(* CODESYS project Lib.library
   Author: Sha
   Placeholder: Lib
   Title: Lib
   Version: 0.1.2
   DefaultNamespace: Lib
   Company: Terza-automation

Project tree, tasks and I/O mapping:
  libraries: CmpBitmapPool, * (System); Tc2_ModbusRTU, * (Beckhoff Automation GmbH); Tc2_Standard, * (Beckhoff Automation GmbH); Tc2_System, * (Beckhoff Automation GmbH); Tc2_Utilities, * (Beckhoff Automation GmbH); Tc3_Module, * (Beckhoff Automation GmbH)
  DUTs/
    data type Beckhoff_AI
    data type ModbusUnion
    data type RealWordUnion
    data type RTU_EM
    data type RTU_STS
    data type RTU_THT
  GVLs/
    global variables GVL
    global variables GVL_DataHalls
    global variables GVL_Electrical
    global variables GVL_EM
    global variables GVL_HW
    global variables GVL_PCS
    global variables GVL_SCS
    global variables GVL_STS
    global variables GVL_THT
  POUs/
    function block AccumDDHHMM [LD]
    function block AccumTimes [LD]
    function AI_OOR [ST]
    function block CAC_Analog [ST]
    function block CAC_Average [ST]
    function block CAC_Mirror [ST]
    function block FB_AI_Scaling [ST]
    function block FB_AO_Scaling [ST]
    program MAIN [ST]
    function block ModbusRTU_EM_Bell [ST]
    function block ModbusRTU_EM_Integra [ST]
    function block ModbusRTU_STS [ST]
    function block ModbusRTU_THT [ST]
    function block OneATS [ST]
    function block OneCRAH [ST]
    function block OneDI [ST]
    function block OneEnergyMeter [ST]
    function block OneFire_Suppr [ST]
    function block OneGen [ST]
    function block OneGLP [ST]
    function block OneIDF [ST]
    function block OneIsolator_Latch [LD]
    function block OnePDU [ST]
    function block OnePumpFF_Latch [LD]
    function block OneSpeed_Override [LD]
    function block OneSTS [ST]
    function block OneSTS_RTU [ST]
    function block OneSWBL [ST]
    function block OneTie_BRK [ST]
    function block OneUPS [ST]
    function block OneVSD_Latch [LD]
    function ReadModbusBool [ST]
    function ReadModbusReal [ST]
    function ReadModusTime [ST]
    function block WriteModbusBool [ST]
    function block WriteModbusReal [ST]
    function block WriteModbusWord [ST]
  Version/
    global variables Global_Version
  VISUs/
    visualisation AminCRAH
    text list CRAH_Isolator_Status
    text list CRAH_Status
    visualisation Dialog_CRAH
    visualisation Dialog_DP_Field
    visualisation Dialog_EnergyMeter
    visualisation Dialog_PDU
    visualisation Dialog_THT_Field
    text list Energy_Meters_Status
    text list Equipment_Status
    text list GLP_Available
    text list GLP_Status
    text list Leak_Detection_Fault
    visualisation Obj_Alarm_Equipment
    visualisation Obj_DP_Field
    visualisation Obj_Energy_Meter
    visualisation Obj_GLP_Avail
    visualisation Obj_GLP_Status
    visualisation Obj_Healthy_Failed_Field
    visualisation Obj_Leak_Detection
    visualisation Obj_PDU_Breaker
    visualisation Obj_PDU_Surge
    visualisation Obj_Terminal
    visualisation Obj_THT_Field
    text list PDU_Breaker_Status
    text list PDU_Surge_Status
  text list GlobalTextList
*)

// DUTs/Beckhoff_AI
TYPE Beckhoff_AI :
STRUCT
	rawValue   : WORD;
	OutOfRange : BOOL;
	Offline    : BOOL;
	Value      : REAL;

END_STRUCT
END_TYPE

// DUTs/ModbusUnion
TYPE ModbusUnion :
UNION
	realValue : REAL;
	longValue : DWORD;
	wordValue : ARRAY[1..2] OF WORD;
	timeValue : TIME;
END_UNION
END_TYPE

// DUTs/RealWordUnion
TYPE RealWordUnion :
UNION
	RealValue: REAL;
	UDINTValue: UDINT;
	WordArray: ARRAY[1..2] OF WORD;
END_UNION
END_TYPE

// DUTs/RTU_EM
TYPE RTU_EM :
STRUCT
	Status: WORD;
	Operating_Hrs: REAL;
	Energy: REAL;
	Volume: REAL;
	Supply_Temp: REAL;
	Return_Temp: REAL;
	Temp_Diff: REAL;
	CommsError: BOOL;
	CommsErrorCode: INT;	
END_STRUCT
END_TYPE

// DUTs/RTU_STS
TYPE RTU_STS :
STRUCT
	CommsError : BOOL;
	CommsErrorCode : INT;

	PRI_VA : REAL;
	PRI_VB : REAL;
	PRI_VC : REAL;
	OTP_VA : REAL;
	OTP_VB : REAL;
	OTP_VC : REAL;
	AMPSA : REAL;
	AMPSB : REAL;
	AMPSC : REAL;
	FREQ : REAL;
	SEC_VA : REAL;
	SEC_VB : REAL;
	SEC_VC : REAL;
	OTP_LOAD_A : REAL;
	OTP_LOAD_B : REAL;
	OTP_LOAD_C : REAL;
	COM_ALM : BOOL;
	OTP_KW_A : REAL;
	OTP_KW_B : REAL;
	OTP_KW_C : REAL;
	OTP_KVA_A : REAL;
	OTP_KVA_B : REAL;
	OTP_KVA_C : REAL;
	PF_A : REAL;
	PF_B : REAL;
	PF_C : REAL;

	OTP_BKR_OPN : BOOL;
	L1_INP_BKR_OPN : BOOL;
	L2_INP_BKR_OPN : BOOL;
	L1_BYP_BKR_TRP : BOOL;
	L2_BYP_BKR_TRP : BOOL;
	OTP_BKR_TRP : BOOL;
	L1_INP_BKR_TRP : BOOL;
	L2_INP_BKR_TRP : BOOL;
	FANS_FAIL : BOOL;
	
END_STRUCT
END_TYPE

// DUTs/RTU_THT
TYPE RTU_THT :
STRUCT
	Temp: REAL;
	RH: REAL;
	Temp_OOR : BOOL;
	RH_OOR : BOOL;
	CommsError : BOOL;
	CommsErrorCode : INT;	
END_STRUCT
END_TYPE

// GVLs/GVL
{attribute 'qualified_only'}
VAR_GLOBAL
	mb_Input_Coils    	:	ARRAY [0..511] OF BOOL;
	mb_Output_Coils 	:   ARRAY [0..511] OF BOOL;
 	mb_Input_Registers 	:   ARRAY [0..511] OF WORD;
 	mb_Output_Registers :   ARRAY [0..255] OF WORD;
	
	nInputCoilIndex: INT;
	nOutputCoilIndex: INT;
	nInputRegisterIndex: INT;
	nOutputRegisterIndex: INT;
END_VAR

// GVLs/GVL_DataHalls
{attribute 'qualified_only'}
VAR_GLOBAL CONSTANT
	StartInputCoilIndex_CRAH : INT := 0;			// uses 0-95
	StartInputCoilIndex_PDU : INT := 120;			// uses 120-295 
	StartInputCoilIndex_CAC : INT := 0;				// not used
	StartInputCoilIndex_IDF : INT := 310;           // uses 310-331
	StartInputCoilIndex_GLP : INT := 350;           // uses 350-361
	StartInputCoilIndex_ATS : INT := 370;           // uses 370-385
	StartInputCoilIndex_OtherDIs : INT := 400;		// uses 400-411
	StartInputCoilIndex_E_METER : INT := 420;		// uses 420-421
	StartInputCoilIndex_IO : INT := 430;			// uses 430-469
    StartInputCoilIndex_RTUStat : INT := 480;		// uses 480-495
	
	StartOutputCoilIndex_CRAH : INT := 0;			// uses 0-31
	StartOutputCoilIndex_PDU : INT := 0;			// not used
	StartOutputCoilIndex_CAC : INT := 80;			// uses 80-447
	StartOutputCoilIndex_OtherDIs : INT := 0;		// not used
	StartoutputCoilIndex_E_METER : INT := 0;		// not used
	StartoutputCoilIndex_IO : INT := 0;				// not used
	StartoutputCoilIndex_IDF : INT := 0;	        // not used
	StartoutputCoilIndex_GLP : INT := 0;	        // not used
	StartoutputCoilIndex_ATS : INT := 60;	        // uses 60-65
	StartOutputCoilIndex_RTUStat : INT := 0;	    // not used
	
	StartInputRegisterIndex_CRAH: INT := 0;			// uses 0-127
	StartInputRegisterIndex_PDU: INT := 0;			// not used
	StartInputRegisterIndex_CAC: INT := 0;			// not used
	StartInputRegisterIndex_OtherDIs : INT := 0;	// not used
	StartInputRegisterIndex_E_METER : INT := 128;	// uses 128-154
    StartInputRegisterIndex_IO : INT := 0;			// not used
	StartInputRegisterIndex_IDF : INT := 0;			// not used
	StartInputRegisterIndex_GLP : INT := 0;			// not used
	StartInputRegisterIndex_ATS : INT := 0;			// not used
	StartInputRegisterIndex_RTUStat : INT := 161;	// uses 161-176 
		
	StartOutputRegisterIndex_CRAH: INT := 0;		// not used
	StartOutputRegisterIndex_PDU: INT := 0;			// not used
	StartOutputRegisterIndex_CAC: INT := 0;			// uses 0-143
	StartOutputRegisterIndex_OtherDIs : INT := 0;	// not used
	StartoutputRegisterIndex_E_METER : INT := 0;	// not used
	StartoutputRegisterIndex_IO : INT := 0;			// not used
	StartoutputRegisterIndex_IDF : INT := 0;		// not used
	StartoutputRegisterIndex_GLP : INT := 0;		// not used
	StartoutputRegisterIndex_ATS : INT := 0;		// not used
	StartOutputRegisterIndex_RTUStat : INT := 0;	// not used
	


END_VAR

// GVLs/GVL_Electrical
{attribute 'qualified_only'}
VAR_GLOBAL CONSTANT
	StartInputCoilIndex_CRAH : INT := 0;			     // uses 0-29
	StartInputCoilIndex_SWBL : INT := 30;			     // uses 30-122 (third & fourth switchboards and STS overlap, but no system has these)
	StartInputCoilIndex_CAC : INT := 0;				     // not used
	StartInputCoilIndex_STS : INT := 98;			     // uses 98-225 no panel has STS and either GLP or ATS
	StartInputCoilIndex_GLP : INT := 210;          		 // uses 210-221
	StartInputCoilIndex_ATS : INT := 222;                // uses 222-244 no panel has ATS and GEN
	StartInputCoilIndex_GEN : INT := 238;			     // uses 238-247
	StartInputCoilIndex_UPS : INT := 248;			     // uses 248-262
	StartInputCoilIndex_TX : INT := 263;			     // uses 263-270
	StartInputCoilIndex_Fire_Suppr : INT := 273;		 // uses 273-296
	StartInputCoilIndex_OtherDIs : INT := 297;		     // uses 297-330
	StartInputCoilIndex_STSRTU : INT := 331;		     // uses 331-407
 	StartInputCoilIndex_IO : INT := 408;				 // uses 408-430
 	StartInputCoilIndex_RTUStat : INT := 431;		 	 // uses 431-440
	StartInputCoilIndex_Tie_BRK : INT := 450;            // uses 450-465
	StartInputCoilIndex_EMG_LIT : INT := 471;			 // uses 471-488
   
	StartOutputCoilIndex_CRAH : INT := 0;			     // uses 0-11
	StartOutputCoilIndex_SWBL : INT := 0;			     // not used
	StartOutputCoilIndex_CAC : INT := 23;			     // uses 23-52
	StartOutputCoilIndex_OtherDIs : INT := 0;		     // not used 
	StartOutputCoilIndex_GEN : INT := 0;	             // not used
	StartOutputCoilIndex_UPS : INT := 0;	             // not used
	StartOutputCoilIndex_TX : INT := 0;				     // not used
	StartOutputCoilIndex_Fire_Suppr : INT := 0;	         // not used
	StartOutputCoilIndex_ATS : INT := 20;	             // uses 20-22
	StartOutputCoilIndex_GLP : INT := 0;	      		 // not used
	StartOutputCoilIndex_Tie_BRK : INT := 0;	         // not used
	StartOutputCoilIndex_STS : INT := 12;	             // uses 12-19
	StartOutputCoilIndex_STSRTU : INT := 0;	             // not used
 	StartOutputCoilIndex_IO : INT := 0;				 	 // not used
 	StartOutputCoilIndex_RTUStat : INT := 0;			 // not used
	StartOutputCoilIndex_EMG_LIT : INT := 0;	         // not used 
	
	StartInputRegisterIndex_CRAH: INT := 0;			     // uses 0-46
	StartInputRegisterIndex_SWBL: INT := 0;			     // not used
	StartInputRegisterIndex_CAC: INT := 0;			     // not used
	StartInputRegisterIndex_OtherDIs : INT := 0;	     // not used
	StartInputRegisterIndex_GEN : INT := 0;			     // not used
	StartInputRegisterIndex_UPS : INT := 0;			     // not used
    StartInputRegisterIndex_TX : INT := 0;			     // not used
	StartInputRegisterIndex_Fire_Suppr : INT := 0;	     // not used
	StartInputRegisterIndex_ATS : INT := 0;			     // not used
	StartInputRegisterIndex_GLP : INT := 0;	    		 // not used
	StartInputRegisterIndex_Tie_BRK : INT := 0;	         // not used
	StartInputRegisterIndex_STS : INT := 0;			     // not used
	StartInputRegisterIndex_STSRTU : INT := 61;			 // uses 61-460
 	StartInputRegisterIndex_IO : INT := 0;				 // not used
 	StartInputRegisterIndex_RTUStat : INT := 47;		 // uses 47-56
	StartInputRegisterIndex_EMG_LIT : INT := 0;			 // not used
		
	StartOutputRegisterIndex_CRAH: INT := 0;		     // not used
	StartOutputRegisterIndex_SWBL: INT := 0;		     // not used
	StartOutputRegisterIndex_CAC: INT := 0;			     // uses 0-10
	StartOutputRegisterIndex_OtherDIs : INT := 0;	     // not used
	StartOutputRegisterIndex_GEN : INT := 0;			 // not used
	StartOutputRegisterIndex_UPS : INT := 0;			 // not used
	StartOutputRegisterIndex_TX : INT := 0;			     // not used
	StartOutputRegisterIndex_Fire_Suppr : INT := 0;	     // not used
	StartOutputRegisterIndex_ATS : INT := 0;		     // not used
	StartOutputRegisterIndex_GLP : INT := 0;			 // not used
	StartOutputRegisterIndex_Tie_BRK : INT := 0;		 // not used
	StartOutputRegisterIndex_STS : INT := 0;			 // not used
	StartOutputRegisterIndex_STSRTU : INT := 0;			 // not used
 	StartOutputRegisterIndex_IO : INT := 0;				 // not used
 	StartOutputRegisterIndex_RTUStat : INT := 0;		 // not used
	StartOutputRegisterIndex_EMG_LIT : INT := 0;	     // not used
	
END_VAR

// GVLs/GVL_EM
{attribute 'qualified_only'}
VAR_GLOBAL
	EM: ARRAY[1..5] OF RTU_EM;
END_VAR

// GVLs/GVL_HW
{attribute 'qualified_only'}
VAR_GLOBAL
	//Date and Time
    fbGetLocalSystemTime: FB_LocalSystemTime;
	sSystemDateTime : STRING;
	sSystemTime : STRING;
	sSystemDate : STRING;	

	// Coupler state - a UINT that should be 8 if its healthy
	CouplerStatus AT %I* : UINT;
	Term02Status AT %I* : WORD;
	Term03Status AT %I* : WORD;
	Term04Status AT %I* : WORD;
	Term05Status AT %I* : WORD;
	Term06Status AT %I* : WORD;
	Term07Status AT %I* : WORD;
	Term08Status AT %I* : WORD;
	Term09Status AT %I* : WORD;
	Term10Status AT %I* : WORD;
	Term11Status AT %I* : WORD;
	Term12Status AT %I* : WORD;
	Term13Status AT %I* : WORD;
	Term14Status AT %I* : WORD;
	Term15Status AT %I* : WORD;
	Term16Status AT %I* : WORD;
	Term17Status AT %I* : WORD;
	Term18Status AT %I* : WORD;
	Term19Status AT %I* : WORD;
	Term20Status AT %I* : WORD;
	Term21Status AT %I* : WORD;
	Term22Status AT %I* : WORD;
	Term23Status AT %I* : WORD;
	Term24Status AT %I* : WORD;
	Term25Status AT %I* : WORD;
	Term26Status AT %I* : WORD;
	Term27Status AT %I* : WORD;
	Term28Status AT %I* : WORD;
	Term29Status AT %I* : WORD;
	Term30Status AT %I* : WORD;
	Term31Status AT %I* : WORD;
	Term32Status AT %I* : WORD;
	Term33Status AT %I* : WORD;
	Term34Status AT %I* : WORD;
	Term35Status AT %I* : WORD;
	Term36Status AT %I* : WORD;
    Term37Status AT %I* : WORD;
    Term38Status AT %I* : WORD;
    Term39Status AT %I* : WORD;
    Term40Status AT %I* : WORD;
	
	// I/O module status
	CouplerOffline : BOOL;
	Term02Offline : BOOL;
	Term03Offline : BOOL;
	Term04Offline : BOOL;
	Term05Offline : BOOL;
	Term06Offline : BOOL;
	Term07Offline : BOOL;
	Term08Offline : BOOL;
	Term09Offline : BOOL;
	Term10Offline : BOOL;
	Term11Offline : BOOL;
	Term12Offline : BOOL;
	Term13Offline : BOOL;
	Term14Offline : BOOL;
	Term15Offline : BOOL;
	Term16Offline : BOOL;
	Term17Offline : BOOL;
	Term18Offline : BOOL;
	Term19Offline : BOOL;
	Term20Offline : BOOL;
	Term21Offline : BOOL;
	Term22Offline : BOOL;
	Term23Offline : BOOL;
	Term24Offline : BOOL;
	Term25Offline : BOOL;
	Term26Offline : BOOL;
	Term27Offline : BOOL;
	Term28Offline : BOOL;
	Term29Offline : BOOL;
	Term30Offline : BOOL;
	Term31Offline : BOOL;
	Term32Offline : BOOL;
	Term33Offline : BOOL;
	Term34Offline : BOOL;
	Term35Offline : BOOL;
	Term36Offline : BOOL;
	Term37Offline : BOOL;
	Term38Offline : BOOL;
	Term39Offline : BOOL;
	Term40Offline : BOOL;
END_VAR

// GVLs/GVL_PCS
{attribute 'qualified_only'}
VAR_GLOBAL
	StartInputCoilIndex_DI: 			INT:=0;		// hardwired DI state sent to OA	
	StartInputCoilIndex_DO: 			INT:=40;	// hardwired DO state sent to OA
	StartInputCoilIndex_TerminalStatus: INT:=50;	// module state sent to OA
	StartInputCoilIndex_AI: 			INT:=100;	// AI OutOfRange status sent to OA
	StartInputCoilIndex_Control:		INT:=200;	// boolean values for control sent by OA
	
	StartOutputCoilIndex_DO: 			INT:=0;		// OA demand for state of digital outputs
	StartOutputCoilIndex_Control:		INT:=200;	// boolean values for control sent to OA
	
	StartInputRegisterIndex_AI: 		INT:=0;		// hardwired AI states sent to OA (each sent as real, using two registers)
    StartInputRegisterIndex_AO:	        INT:=50;	// hardwired AI states sent to OA (each sent as real, using two registers)
	StartInputRegisterIndex_Control:	INT:=200;	// integer and real values for control sent by OA

	StartOutputRegisterIndex_AO: 		INT:=0;		// OA demand for states of analog outputs
	StartOutputRegisterIndex_Control:	INT:=200;	// integer and real values for control sent to OA
END_VAR

// GVLs/GVL_SCS
{attribute 'qualified_only'}
VAR_GLOBAL
	
	StartInputCoilIndex_DI: 			INT:=0;		// hardwired DI state sent to OA	
	StartInputCoilIndex_DO: 			INT:=40;	// hardwired DO state sent to OA
	StartInputCoilIndex_TerminalStatus: INT:=50;	// module state sent to OA
	StartInputCoilIndex_AI: 			INT:=100;	// AI OutOfRange status sent to OA
	StartInputCoilIndex_RTUStat:		INT:=150;	// RTU comms status 
	StartInputCoilIndex_Control:		INT:=200;	// boolean values for control sent by OA
	StartInputCoilIndex_E_Meter:		INT:=250;	// Energy meter comms status
	
	StartOutputCoilIndex_DO: 			INT:=0;		// OA demand for state of digital outputs
	StartOutputCoilIndex_RTUStat:		INT:= 0;	// not used
	StartOutputCoilIndex_Control:		INT:=200;	// boolean values for control sent to OA
	StartOutputCoilIndex_E_Meter:		INT:= 0;	// not used
	
	StartInputRegisterIndex_AI: 		INT:=0;		// hardwired AI states sent to OA (each sent as real, using two registers)
    StartInputRegisterIndex_AO:	        INT:=50;	// hardwired AI states sent to OA (each sent as real, using two registers)
	StartInputRegisterIndex_RTUStat:	INT:=150;	// RTU comms error codes 
	StartInputRegisterIndex_Control:	INT:=200;	// integer and real values for control sent by OA
	StartInputRegisterIndex_E_Meter:	INT:=250;	// Energy meter data 

	StartOutputRegisterIndex_AO: 		INT:=0;		// OA demand for states of analog outputs
	StartOutputRegisterIndex_RTUStat:	INT:= 0;	// not used
	StartOutputRegisterIndex_Control:	INT:=200;	// integer and real values for control sent to OA
	StartOutputRegisterIndex_E_Meter:	INT:= 0;	// not used

END_VAR

// GVLs/GVL_STS
{attribute 'qualified_only'}
VAR_GLOBAL
	STS : ARRAY [1..10] OF RTU_STS;
END_VAR

// GVLs/GVL_THT
{attribute 'qualified_only'}
VAR_GLOBAL
	THT : ARRAY [1..14] OF RTU_THT;
END_VAR

VAR_GLOBAL CONSTANT
	Temp_OOR_Min : REAL :=   0.0;
	Temp_OOR_Max : REAL :=  50.0;
	RH_OOR_Min   : REAL :=   0.0;
	RH_OOR_Max   : REAL := 100.0;
END_VAR

// Version/Global_Version
{attribute 'TcGenerated'}
{attribute 'no-analysis'}
{attribute 'linkalways'}
// This function has been automatically generated from the project information.
VAR_GLOBAL CONSTANT
	{attribute 'const_non_replaced'}
	stLibVersion_Lib : ST_LibVersion := (iMajor := 0, iMinor := 1, iBuild := 2, iRevision := 0, nFlags := 0, sVersion := '0.1.2');
END_VAR

// POUs/AccumDDHHMM
FUNCTION_BLOCK AccumDDHHMM
VAR_INPUT
	State: BOOL;
	Retentive: BOOL;
	Reset:BOOL;
END_VAR

VAR PERSISTENT
	Mins: WORD;
	Hrs:  WORD;
	Days: WORD;	
END_VAR
VAR
	DisplayTime: STRING;
	timer: TON;
	timerPT: TIME:= T#1M;
	StateToOff: F_TRIG;
END_VAR

VAR_TEMP
	displayTimeFormat: FB_FormatString;
END_VAR
VAR // added by the converter: edge detectors and wires of the graphical bodies
    _w1, _w2, _w3, _w4 : BOOL;
END_VAR

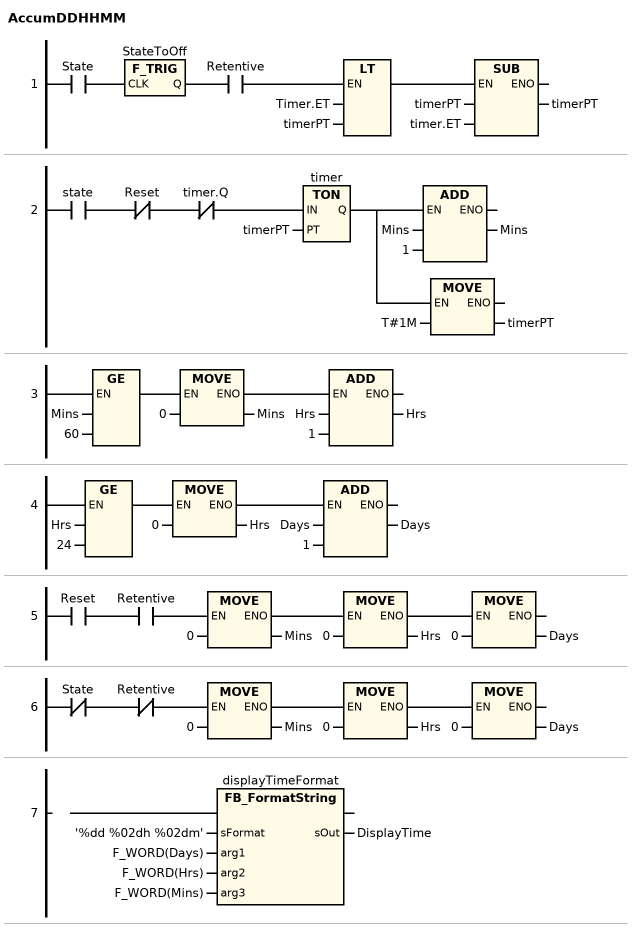
// NETWORK 1
StateToOff(CLK := State); // F_TRIG
IF StateToOff.Q AND Retentive AND Timer.ET < timerPT THEN timerPT := timerPT - timer.ET; END_IF

// NETWORK 2
timer(IN := state AND NOT Reset AND NOT timer.Q, PT := timerPT); // TON
IF timer.Q THEN Mins := Mins + 1; END_IF
IF timer.Q THEN timerPT := T#1M; END_IF

// NETWORK 3
_w1 := Mins >= 60;
IF _w1 THEN Mins := 0; END_IF
IF _w1 THEN Hrs := Hrs + 1; END_IF

// NETWORK 4
_w2 := Hrs >= 24;
IF _w2 THEN Hrs := 0; END_IF
IF _w2 THEN Days := Days + 1; END_IF

// NETWORK 5
_w3 := Reset AND Retentive;
IF _w3 THEN Mins := 0; END_IF
IF _w3 THEN Hrs := 0; END_IF
IF _w3 THEN Days := 0; END_IF

// NETWORK 6
_w4 := NOT State AND NOT Retentive;
IF _w4 THEN Mins := 0; END_IF
IF _w4 THEN Hrs := 0; END_IF
IF _w4 THEN Days := 0; END_IF

// NETWORK 7
displayTimeFormat(
    sFormat := '%dd %02dh %02dm',
    arg1 := F_WORD(Days),
    arg2 := F_WORD(Hrs),
    arg3 := F_WORD(Mins),
    sOut => DisplayTime); // FB_FormatString

END_FUNCTION_BLOCK

// POUs/AccumTimes
FUNCTION_BLOCK AccumTimes
VAR_INPUT
	State: BOOL;	
END_VAR

VAR PERSISTENT
	Num : WORD;
	ResetAccum: BOOL;

	cntOn: CTU;
	Accum: AccumDDHHMM;
	On: AccumDDHHMM;
	Off: AccumDDHHMM;
END_VAR

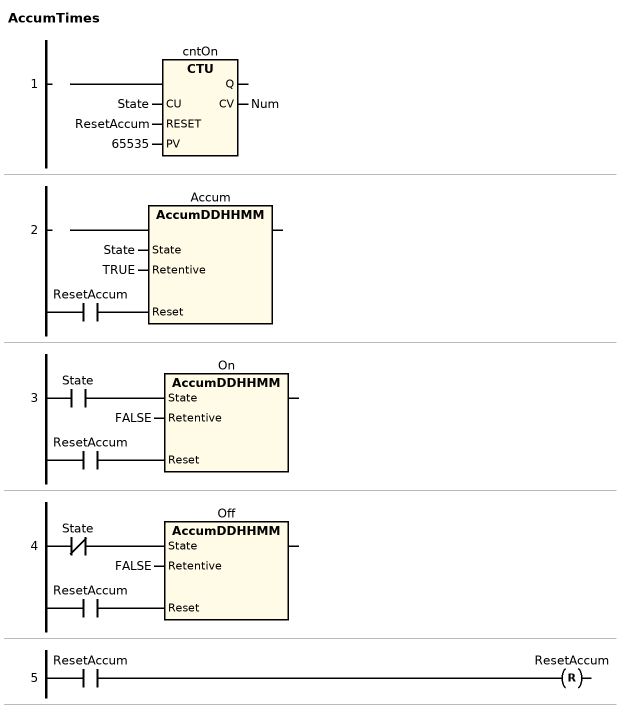
// NETWORK 1
cntOn(CU := State, RESET := ResetAccum, PV := 65535, CV => Num); // CTU

// NETWORK 2
Accum(State := State, Retentive := TRUE, Reset := ResetAccum); // AccumDDHHMM

// NETWORK 3
On(State := State, Retentive := FALSE, Reset := ResetAccum); // AccumDDHHMM

// NETWORK 4
Off(State := NOT State, Retentive := FALSE, Reset := ResetAccum); // AccumDDHHMM

// NETWORK 5
ResetAccum R= ResetAccum;

END_FUNCTION_BLOCK

// POUs/AI_OOR
FUNCTION AI_OOR : bool
VAR_INPUT
	Status: WORD;
END_VAR

// calculate whether the status for an analog input is indicating an error
// the error bit is the 7th bit of the status word
// access to bits is base 0, so the 7th bit is accessed with index 6

AI_OOR:= Status.6;

END_FUNCTION

// POUs/CAC_Analog
FUNCTION_BLOCK CAC_Analog
VAR_INPUT
	Value: REAL;
	OutOfRange : BOOL;
	Offline: BOOL;
END_VAR
VAR
	SetInclude: BOOL;
	SetExclude : BOOL;
	Excluded: BOOL;
	Alarm : BOOL;
	SetIncludeTrig: R_TRIG;
	SetExcludeTrig: R_TRIG;
END_VAR

VAR_TEMP
	i:INT;
	modbusReal: ModbusUnion;
END_VAR


i:= GVL.nOutputRegisterIndex;
modbusReal.realValue:= Value;
GVL.mb_Output_Registers[i+0]:= modbusReal.wordValue[1];
GVL.mb_Output_Registers[i+1]:= modbusReal.wordValue[2];
GVL.nOutputRegisterIndex:=i+2;

i:= GVL.nOutputCoilIndex;
GVL.mb_Output_Coils[i]:= OutOfRange;
GVL.mb_Output_Coils[i+1]:= Offline;

SetIncludeTrig(CLK:= SetInclude);
IF SetIncludeTrig.Q THEN 
	GVL.mb_Output_Coils[i+2]:= TRUE;
ELSIF SetInclude AND GVL.mb_Output_Coils[i+2] = FALSE THEN
 	SetInclude:=FALSE;
END_IF


SetExcludeTrig(CLK:=SetExclude);
IF SetExcludeTrig.Q THEN 
	GVL.mb_Output_Coils[i+3]:= TRUE;	
ELSIF SetExclude AND GVL.mb_Output_Coils[i+3]= FALSE THEN 
	SetExclude:=FALSE;
END_IF


Excluded:= GVL.mb_Output_Coils[i+4];
Alarm:= GVL.mb_Output_Coils[i+5];

GVL.nOutputCoilIndex:= i + 6;

END_FUNCTION_BLOCK

// POUs/CAC_Average
FUNCTION_BLOCK CAC_Average
VAR_INPUT
END_VAR
VAR_OUTPUT
END_VAR
VAR
	Value: REAL;
	Alarm: BOOL;
	OutOfRange: BOOL;
	Offline: BOOL;
END_VAR

VAR_TEMP
	i: INT;
	modbusReal: ModbusUnion;
END_VAR


i:= GVL.nOutputRegisterIndex;
modbusReal.wordValue[1]:= GVL.mb_Output_Registers[i+0];
modbusReal.wordValue[2]:= GVL.mb_Output_Registers[i+1];

Value:= modbusReal.realValue;
GVL.nOutputRegisterIndex:= i+2;


i:= GVL.nOutputCoilIndex;
OutOfRange:= FALSE;
Offline:= GVL.mb_Output_Coils[i+0];
Alarm:= GVL.mb_Output_Coils[i+1];
GVL.nOutputCoilIndex:= i+2;

END_FUNCTION_BLOCK

// POUs/CAC_Mirror
FUNCTION_BLOCK CAC_Mirror
VAR
	Value: REAL;
	OutOfRange: BOOL;
	Offline: BOOL;
	SetInclude: BOOL;
	SetExclude: BOOL;
	Excluded: BOOL;
	Alarm: BOOL;
	SetIncludeTrig: R_TRIG;
	SetExcludeTrig: R_TRIG;
END_VAR

VAR_TEMP
	i:INT;
	modbusReal: ModbusUnion;
END_VAR


i:= GVL.nOutputRegisterIndex;
modbusReal.wordValue[1]:= GVL.mb_Output_Registers[i+0];
modbusReal.wordValue[2]:= GVL.mb_Output_Registers[i+1];
Value:= modbusReal.realValue;
GVL.nOutputRegisterIndex:= i+2;

i:= GVL.nOutputCoilIndex;
OutOfRange:= GVL.mb_Output_Coils[i+0];
Offline:= GVL.mb_Output_Coils[i+1];

SetIncludeTrig(CLK:=SetInclude);

IF SetIncludeTrig.Q THEN 
	GVL.mb_Output_Coils[i+2] := TRUE;
ELSIF SetInclude AND GVL.mb_Output_Coils[i+2]= FALSE THEN 
	SetInclude:= FALSE;
END_IF

SetExcludeTrig(CLK:= SetExclude);
	
IF SetExcludeTrig.Q THEN 
	GVL.mb_Output_Coils[i+3] := TRUE;
ELSIF SetExclude AND GVL.mb_Output_Coils[i+3]= FALSE THEN 
	SetExclude:= FALSE;
END_IF


Excluded:= GVL.mb_Output_Coils[i+4];
Alarm:= GVL.mb_Output_Coils[i+5];
GVL.nOutputCoilIndex:= i+6;

END_FUNCTION_BLOCK

// POUs/FB_AI_Scaling
FUNCTION_BLOCK FB_AI_Scaling
VAR_INPUT
	I_Input: INT;
	I_Input_Min:  REAL :=0;
	I_Input_Max:  REAL :=100;
	I_Output_Min: REAL :=0;
	I_Output_Max: REAL :=3;
END_VAR
VAR_OUTPUT
	O_Output:REAL;
	O_Error:BOOL;	
END_VAR
VAR
	L_Input:INT;
END_VAR

VAR_TEMP
	i:INT;
	modbusReal: ModbusUnion;
END_VAR


IF I_Input_Max <> 0 AND I_Output_Max <> 0 THEN 
	IF I_Input_Min <= I_Input_Max THEN 
		L_Input:=I_Input;
		O_Output:= ((I_Output_Max - I_Output_Min) / (I_Input_Max - I_Input_Min) * (I_input - I_Input_Min) + I_Output_Min);
		O_Error:=FALSE;
	ELSE
		I_Input:= L_Input;	
	END_IF
ELSE
	O_Error:=TRUE;
END_IF


i:=GVL.nInputRegisterIndex;
modbusReal.realValue:= O_Output;
GVL.mb_Input_Registers[i+0]:= modbusReal.wordValue[1];
GVL.mb_Input_Registers[i+1]:= modbusReal.wordValue[2];
GVL.nInputRegisterIndex:=i+2;

END_FUNCTION_BLOCK

// POUs/FB_AO_Scaling
FUNCTION_BLOCK FB_AO_Scaling
VAR_INPUT
	I_Input:REAL;
	I_Input_Min:REAL:=0;
	I_Input_Max:REAL:=100;
	I_Output_Min:REAL :=0;
	I_Output_Max:REAL :=0;
END_VAR

VAR_OUTPUT
	O_Output: INT;
	O_Error: BOOL;
END_VAR

VAR
	L_Input:REAL;
END_VAR

VAR_TEMP
	i:INT;
	modbusReal: ModbusUnion;
END_VAR


IF I_Input_Max <> 0 AND I_Output_Max <> 0 THEN 
	IF I_Input <=I_Input_Max THEN 	
		L_Input:= I_Input;
		O_Output:= REAL_TO_INT((I_Output_Max - I_Output_Min) / (I_Input_Max - I_Input_Min) * (I_input - I_Input_Min) + I_Output_Min);
		O_Error:= FALSE;	
	ELSE
		I_Input:= L_Input;	
	END_IF
ELSE	
	O_Error:= TRUE;
END_IF

i:= GVL.nInputRegisterIndex;
modbusReal.realValue := L_Input;
GVL.mb_Input_Registers[i+0] := modbusReal.WordValue[1];
GVL.mb_Input_Registers[i+1] := modbusReal.WordValue[2];
GVL.nInputRegisterIndex := i+2;

END_FUNCTION_BLOCK

// POUs/MAIN
PROGRAM MAIN
VAR
END_VAR

END_PROGRAM

// POUs/ModbusRTU_EM_Bell
FUNCTION_BLOCK ModbusRTU_EM_Bell
VAR_INPUT
	MB_FirstUnitID: BYTE;
	MB_LastUnitID:  BYTE;
	EM_First: INT := 1;
END_VAR
VAR_OUTPUT
END_VAR
VAR
END_VAR

END_FUNCTION_BLOCK

// POUs/ModbusRTU_EM_Integra
FUNCTION_BLOCK ModbusRTU_EM_Integra
VAR_INPUT
	MB_FirstUnitID: BYTE;
	MB_LastUnitID: BYTE;
	EM_First: INT := 1;
END_VAR

VAR
	ModbusTerm: ModbusRtuMaster_KL6x22B;
	
	MB_UnitID : BYTE := 0;
	MB_Address : WORD := 0;
	MB_Quantity : WORD := 2;
	MB_ReadData : ModbusUnion;

	MB_TrigRead : BOOL := FALSE;
	MB_CommState: (TRIGGER, TRIGGERED, WAIT_RESPONSE, SETUP_NEXT_MESSAGE) := TRIGGER;
	tmrDelay: TON;
END_VAR


VAR CONSTANT
	MODBUS_DELAY : TIME := T#100MS;
END_VAR

VAR	
	EMNum: INT;
	MessageNum: INT;
END_VAR

IF (MB_UnitID < MB_FirstUnitID) THEN
	MB_UnitID := MB_FirstUnitID;
	EMNum := EM_First;
	MessageNum := 1;
	MB_Address := 0;
END_IF

IF (MB_UnitID > MB_LastUnitID) THEN
	MB_UnitID := MB_FirstUnitID;
	EMNum := EM_First;
	MessageNum := 1;
	MB_Address := 0;
END_IF

ModbusTerm.ReadRegs(
	UnitID:= MB_UnitID, 
	Quantity:= MB_Quantity, 
	MBAddr:= MB_Address, 
	cbLength:= SIZEOF(MB_ReadData), 
	pMemoryAddr:= ADR(MB_ReadData), 
	Execute:= MB_TrigRead, 
	Timeout:= T#1S, 
	BUSY=> , 
	Error=> , 
	ErrorID=> , 
	cbRead=> );
	
	
CASE MB_CommState OF
	TRIGGER:
		tmrDelay(IN:=TRUE, PT:=MODBUS_DELAY);
		IF tmrDelay.Q THEN
			MB_TrigRead := TRUE;
			MB_CommState := TRIGGERED;
		END_IF

	TRIGGERED:
		tmrDelay(IN:=FALSE, PT:=MODBUS_DELAY);
		MB_TrigRead := FALSE;
		MB_CommState := WAIT_RESPONSE;

	WAIT_RESPONSE:
		IF NOT ModbusTerm.BUSY THEN
			GVL_EM.EM[EMNum].CommsError     := ModbusTerm.Error;
			GVL_EM.EM[EMNum].CommsErrorCode := ModbusTerm.ErrorId;
			IF NOT ModbusTerm.Error THEN
				IF MessageNum = 1 THEN
					GVL_EM.EM[EMNum].Status := MB_ReadData.wordValue[2];
				ELSIF MessageNum = 2 THEN
					GVL_EM.EM[EMNum].Operating_Hrs := MB_ReadData.realValue;
				ELSIF MessageNum = 3 THEN
					GVL_EM.EM[EMNum].Energy := MB_ReadData.realValue;
				ELSIF MessageNum = 4 THEN
					GVL_EM.EM[EMNum].Volume := MB_ReadData.realValue;
				ELSIF MessageNum = 5 THEN
					GVL_EM.EM[EMNum].Supply_Temp := MB_ReadData.realValue;
				ELSIF MessageNum = 6 THEN
					GVL_EM.EM[EMNum].Return_Temp := MB_ReadData.realValue;
				ELSIF MessageNum = 7 THEN
					GVL_EM.EM[EMNum].Temp_Diff := MB_ReadData.realValue;
 				END_IF
 
			END_IF
			
			MB_CommState := SETUP_NEXT_MESSAGE;
		END_IF

	SETUP_NEXT_MESSAGE:
		MessageNum := MessageNum + 1;
		IF MessageNum > 7 THEN
			MessageNum := 1;
			MB_UnitID := MB_UnitID + 1;
			EMNum := EMNum + 1;
		END_IF

		IF MessageNum = 1 THEN
			MB_Address := 0;	// read status in word 2
		ELSIF MessageNum = 2 THEN
			MB_Address := 6;	// read operating hours
		ELSIF MessageNum = 3 THEN
			MB_Address := 100;	// read energy
		ELSIF MessageNum = 4 THEN
			MB_Address := 200;	// read volume
		ELSIF MessageNum = 5 THEN
			MB_Address := 800;	// read supply temperature
		ELSIF MessageNum = 6 THEN
			MB_Address := 810;	// read return temperature
		ELSIF MessageNum = 7 THEN
			MB_Address := 820;	// read temperature difference
		END_IF
	
		MB_CommState := TRIGGER;
END_CASE

END_FUNCTION_BLOCK

// POUs/ModbusRTU_STS
FUNCTION_BLOCK ModbusRTU_STS
VAR_INPUT
	MB_FirstUnitID: BYTE;
	MB_LastUnitID: BYTE;
END_VAR
VAR_OUTPUT
END_VAR
VAR
	ModbusTerm: ModbusRtuMaster_KL6x22B;
	
	MB_UnitID : BYTE := 0;
	MB_ReadData : ARRAY[1..71] OF WORD;

	MB_TrigRead : BOOL := FALSE;
	MB_CommState: (TRIGGER, TRIGGERED, WAIT_RESPONSE, SETUP_NEXT_MESSAGE) := TRIGGER;
	tmrDelay: TON;
END_VAR
	
VAR	
	STSNum: INT;
END_VAR


VAR CONSTANT
	MB_Address : WORD := 1;
	MB_Quantity : WORD := 71;

	MODBUS_DELAY : TIME := T#10MS;
END_VAR

IF (MB_UnitID < MB_FirstUnitID) THEN
	MB_UnitID := MB_FirstUnitID;
	STSNum := 1;
END_IF

IF (MB_UnitID > MB_LastUnitID) THEN
	MB_UnitID := MB_FirstUnitID;
	STSNum := 1;
END_IF

ModbusTerm.ReadRegs (
	UnitID:= MB_UnitID, 
	Quantity:= MB_Quantity, 
	MBAddr:= MB_Address - 1, 
	cbLength:= SIZEOF(MB_ReadData), 
	pMemoryAddr:= ADR(MB_ReadData), 
	Execute:= MB_TrigRead, 
	Timeout:= T#1S, 
	BUSY=> , 
	Error=> , 
	ErrorID=> , 
	cbRead=> );
	
CASE MB_CommState OF
	TRIGGER:
		tmrDelay(IN:=TRUE, PT:=MODBUS_DELAY);
		IF tmrDelay.Q THEN
			MB_TrigRead := TRUE;
			MB_CommState := TRIGGERED;
		END_IF

	TRIGGERED:
		tmrDelay(IN:=FALSE, PT:=MODBUS_DELAY);
		MB_TrigRead := FALSE;
		MB_CommState := WAIT_RESPONSE;

	WAIT_RESPONSE:
		IF NOT ModbusTerm.BUSY THEN
			GVL_STS.STS[STSNum].CommsError     := ModbusTerm.Error;
			GVL_STS.STS[STSNum].CommsErrorCode := ModbusTerm.ErrorId;
			IF NOT ModbusTerm.Error THEN
//				IF MessageNum = 1 THEN	// extracts the values in 13 registers #1-13
					GVL_STS.STS[STSNum].PRI_VA := WORD_TO_REAL(MB_ReadData[1]);
					GVL_STS.STS[STSNum].PRI_VB := WORD_TO_REAL(MB_ReadData[2]);
					GVL_STS.STS[STSNum].PRI_VC := WORD_TO_REAL(MB_ReadData[3]);
					GVL_STS.STS[STSNum].OTP_VA := WORD_TO_REAL(MB_ReadData[4]);
					GVL_STS.STS[STSNum].OTP_VB := WORD_TO_REAL(MB_ReadData[5]);
					GVL_STS.STS[STSNum].OTP_VC := WORD_TO_REAL(MB_ReadData[6]);
					GVL_STS.STS[STSNum].AMPSA  := WORD_TO_REAL(MB_ReadData[7]);
					GVL_STS.STS[STSNum].AMPSB  := WORD_TO_REAL(MB_ReadData[8]);
					GVL_STS.STS[STSNum].AMPSC  := WORD_TO_REAL(MB_ReadData[9]);
					GVL_STS.STS[STSNum].FREQ   := WORD_TO_REAL(MB_ReadData[10]);
					GVL_STS.STS[STSNum].SEC_VA := WORD_TO_REAL(MB_ReadData[11]);
					GVL_STS.STS[STSNum].SEC_VB := WORD_TO_REAL(MB_ReadData[12]);
					GVL_STS.STS[STSNum].SEC_VC := WORD_TO_REAL(MB_ReadData[13]);

//				ELSIF MessageNum = 2 THEN	// extracts the values in 3 registers #17-19
					GVL_STS.STS[STSNum].OTP_LOAD_A := WORD_TO_REAL(MB_ReadData[17]);
					GVL_STS.STS[STSNum].OTP_LOAD_B := WORD_TO_REAL(MB_ReadData[18]);
					GVL_STS.STS[STSNum].OTP_LOAD_C := WORD_TO_REAL(MB_ReadData[19]);

//				ELSIF MessageNum = 3 THEN	// extracts the alarms - 4 registers #41-44
					// common alarm is bit 15 of register 41
					GVL_STS.STS[STSNum].COM_ALM :=MB_ReadData[41].15;
					// other alarms of interest are in register 43 
					GVL_STS.STS[STSNum].OTP_BKR_OPN    := MB_ReadData[43].0;
					GVL_STS.STS[STSNum].L1_INP_BKR_OPN := MB_ReadData[43].1;
					GVL_STS.STS[STSNum].L2_INP_BKR_OPN := MB_ReadData[43].2;
					GVL_STS.STS[STSNum].L1_BYP_BKR_TRP := MB_ReadData[43].3;
					GVL_STS.STS[STSNum].L2_BYP_BKR_TRP := MB_ReadData[43].4;
					GVL_STS.STS[STSNum].OTP_BKR_TRP    := MB_ReadData[43].5;
					GVL_STS.STS[STSNum].L1_INP_BKR_TRP := MB_ReadData[43].6;
					GVL_STS.STS[STSNum].L2_INP_BKR_TRP := MB_ReadData[43].7;
					GVL_STS.STS[STSNum].FANS_FAIL      := MB_ReadData[43].8;

//				ELSIF MessageNum = 4 THEN	// extracts the values in 6 registers #56-61
					GVL_STS.STS[STSNum].OTP_KW_A  := WORD_TO_REAL(MB_ReadData[56]) / 10.0;
					GVL_STS.STS[STSNum].OTP_KW_B  := WORD_TO_REAL(MB_ReadData[57]) / 10.0;
					GVL_STS.STS[STSNum].OTP_KW_C  := WORD_TO_REAL(MB_ReadData[58]) / 10.0;
					GVL_STS.STS[STSNum].OTP_KVA_A := WORD_TO_REAL(MB_ReadData[59]) / 10.0;
					GVL_STS.STS[STSNum].OTP_KVA_B := WORD_TO_REAL(MB_ReadData[60]) / 10.0;
					GVL_STS.STS[STSNum].OTP_KVA_C := WORD_TO_REAL(MB_ReadData[61]) / 10.0;

//				ELSIF MessageNum = 5 THEN	// extracts the values in 3 registers #69-71
					GVL_STS.STS[STSNum].PF_A := WORD_TO_REAL(MB_ReadData[69]) / 100.0;
					GVL_STS.STS[STSNum].PF_B := WORD_TO_REAL(MB_ReadData[70]) / 100.0;
					GVL_STS.STS[STSNum].PF_C := WORD_TO_REAL(MB_ReadData[71]) / 100.0;
// 				END_IF
 			END_IF
			
			MB_CommState := SETUP_NEXT_MESSAGE;
		END_IF

	SETUP_NEXT_MESSAGE:
		MB_UnitID := MB_UnitID + 1;
		STSNum := STSNum + 1;
	
		MB_CommState := TRIGGER;
END_CASE

END_FUNCTION_BLOCK

// POUs/ModbusRTU_THT
FUNCTION_BLOCK ModbusRTU_THT
VAR_INPUT
	MB_FirstUnitID: BYTE;
	MB_LastUnitID: BYTE;
END_VAR
VAR_OUTPUT
END_VAR
VAR
	ModbusTerm: ModbusRtuMasterV2_KL6x22B;
	
	MB_UnitID:   BYTE := 0;
	MB_Address:  WORD := 25;
	MB_Quantity: WORD := 4;
	MB_ReadData: ARRAY[1..2] OF ModbusUnion;
	
	MB_TrigRead: BOOL :=FALSE;
	MB_CommState: (TRIGGER, TRIGGERED, WAIT_RESPONSE):=TRIGGER;
	tmrDelay: TON;
END_VAR

IF MB_UnitID < MB_FirstUnitID THEN 
	MB_UnitID:= MB_FirstUnitID;
END_IF

IF MB_UnitID > MB_LastUnitID THEN 
	MB_UnitID:= MB_FirstUnitID;
END_IF

ModbusTerm.ReadRegs(
	UnitID:= MB_UnitID, 
	Quantity:= MB_Quantity, 
	MBAddr:= MB_Address, 
	cbLength:= SIZEOF(MB_ReadData), 
	pMemoryAddr:= ADR(MB_ReadData),  
	Execute:= MB_TrigRead, 
	Timeout:= T#2S, 
	BUSY=> , 
	Error=> , 
	ErrorId=> , 
	cbRead=> );
	
CASE MB_CommState OF 
	TRIGGER:
		tmrDelay(in:=TRUE, PT:=T#1S);
		IF tmrDelay.Q THEN
			MB_TrigRead:=TRUE;
			MB_CommState:=TRIGGERED;
		END_IF
		
	TRIGGERED:
		tmrDelay(in:=FALSE, PT:=T#1S);
		MB_TrigRead:=FALSE;
		MB_CommState:=WAIT_RESPONSE;
		
	WAIT_RESPONSE:
		IF NOT ModbusTerm.BUSY THEN 
			GVL_THT.THT[MB_UnitID].CommsError:= ModbusTerm.Error;
			GVL_THT.THT[MB_UnitID].CommsErrorCode:= ModbusTerm.ErrorId;
			
			IF NOT ModbusTerm.Error THEN 
				GVL_THT.THT[MB_UnitID].Temp:= MB_ReadData[1].realValue;
				GVL_THT.THT[MB_UnitID].RH  := MB_ReadData[2].realValue;
				
				
				GVL_THT.THT[MB_UnitID].Temp_OOR:= (GVL_THT.THT[MB_UnitID].Temp < GVL_THT.Temp_OOR_Min) OR 
												  (GVL_THT.THT[MB_UnitID].Temp > GVL_THT.Temp_OOR_Max);
												  
				GVL_THT.THT[MB_UnitID].Rh_OOR:= (GVL_THT.THT[MB_UnitID].RH < GVL_THT.RH_OOR_Min) OR 
												(GVL_THT.THT[MB_UnitID].RH > GVL_THT.RH_OOR_Max);		   
				
			END_IF
		
			MB_UnitID := MB_UnitID + 1;
			MB_CommState := TRIGGER;
	
		END_IF
END_CASE

END_FUNCTION_BLOCK

// POUs/OneATS
FUNCTION_BLOCK OneATS
VAR_INPUT
	ATS_Avai: BOOL;
	ATS_Avai_Offline : BOOL;
	ATS_SP1 : BOOL;
	ATS_SP1_Offline : BOOL;
	ATS_SP2 : BOOL;
	ATS_SP2_Offline : BOOL;
	ATS_SP0 : BOOL;
	ATS_SP0_Offline : BOOL;
END_VAR
VAR_OUTPUT
	
	Net_Priority : BOOL;
	Source_Priority : BOOL;
	Inhibited: BOOL;
	
END_VAR

VAR_TEMP
	i: INT;
END_VAR

i := GVL.nInputCoilIndex;

GVL.mb_Input_Coils[i+0] := ATS_Avai;
GVL.mb_Input_Coils[i+1] := ATS_Avai_Offline;

GVL.mb_Input_Coils[i+2] := ATS_SP1;
GVL.mb_Input_Coils[i+3] := ATS_SP1_Offline;

GVL.mb_Input_Coils[i+4] := ATS_SP2;
GVL.mb_Input_Coils[i+5] := ATS_SP2_Offline;

GVL.mb_Input_Coils[i+6] := ATS_SP0;
GVL.mb_Input_Coils[i+7] := ATS_SP0_Offline;

GVL.nInputCoilIndex := i + 8;

i:= GVL.nOutputCoilIndex;

Net_Priority := GVL.mb_Output_Coils[i+0];
Source_Priority :=  GVL.mb_Output_Coils[i+1];
Inhibited := GVL.mb_Output_Coils[i+2];

GVL.nOutputCoilIndex := i +3;

END_FUNCTION_BLOCK

// POUs/OneCRAH
FUNCTION_BLOCK OneCRAH
VAR_INPUT
	Running: BOOL;
	Alarm: BOOL;
	Iso1_1_Sts: BOOL;
	Iso1_2_Sts: BOOL;
	Offline: BOOL;	
END_VAR

VAR_OUTPUT
	Enable: BOOL;	
END_VAR

VAR PERSISTENT
	Maintenance: BOOL;
	Inhibited: BOOL;
	HOA: WORD;
	Run: AccumTimes;
	Alm: AccumTimes;
	Ena: AccumTimes;
END_VAR

VAR_TEMP
	i: INT;
	modbusReal: ModbusUnion; 
END_VAR

Run(State:= Running);
Alm(State:= Alarm);
Ena(State:= Enable);

i:= GVL.nInputCoilIndex;

GVL.mb_Input_Coils[i+0] :=  Running;
GVL.mb_Input_Coils[i+1] :=  Alarm;
GVL.mb_Input_Coils[i+2] :=  Offline;
GVL.mb_Input_Coils[i+3] :=  Iso1_1_Sts;
GVL.mb_Input_Coils[i+4] :=  Iso1_2_Sts;

GVL.nInputCoilIndex := i + 5;


i:=GVL.nOutputCoilIndex;

Enable:= GVL.mb_Output_Coils[i+0];
Inhibited:= GVL.mb_Output_Coils[i+1];

GVL.nOutputCoilIndex:= i + 2;

i:= GVL.nInputRegisterIndex;
GVL.mb_Input_Registers[i+0]:= HOA;
GVL.mb_Input_Registers[i+1]:= Run.Num;


modbusReal.realValue:= WORD_TO_REAL(Run.Accum.Days) * 24.0 +
					   WORD_TO_REAL(Run.Accum.Hrs) * 1.0 + 
					   WORD_TO_REAL(Run.Accum.Mins) / 60.0;

GVL.mb_Input_Registers[i+2]:= modbusReal.wordValue[1];
GVL.mb_Input_Registers[i+3]:= modbusReal.wordValue[2];	

modbusReal.realValue:= WORD_TO_REAL(Run.On.Days) * 24.0 +
					   WORD_TO_REAL(Run.On.Hrs) * 1.0 + 
					   WORD_TO_REAL(Run.On.Mins) / 60.0;

GVL.mb_Input_Registers[i+4]:= modbusReal.wordValue[1];
GVL.mb_Input_Registers[i+5]:= modbusReal.wordValue[2];

modbusReal.realValue:= WORD_TO_REAL(Run.Off.Days) * 24.0 +
					   WORD_TO_REAL(Run.Off.Hrs) * 1.0 + 
					   WORD_TO_REAL(Run.Off.Mins) / 60.0;

GVL.mb_Input_Registers[i+6]:= modbusReal.wordValue[1];
GVL.mb_Input_Registers[i+7]:= modbusReal.wordValue[2];	   

						
GVL.nInputRegisterIndex:= i + 8;

END_FUNCTION_BLOCK

// POUs/OneDI
FUNCTION_BLOCK OneDI
VAR_INPUT
	Value: BOOL;
	Offline: BOOL;	
END_VAR

VAR_TEMP
	i:INT;
	
END_VAR


i:=GVL.nInputCoilIndex;

GVL.mb_Input_Coils[i+0]:= Value;
GVL.mb_Input_Coils[i+1]:= Offline;

GVL.nInputCoilIndex:=i+2;

END_FUNCTION_BLOCK

// POUs/OneEnergyMeter
FUNCTION_BLOCK OneEnergyMeter
VAR_INPUT
	Status: WORD;
	Operating_Hrs: REAL;
	Energy: REAL;
	Volume: REAL;
	Supply_Temp: REAL;
	Return_Temp: REAL;
	Temp_Diff: REAL;
	Offline: BOOL;

END_VAR

VAR_TEMP
	i:INT;
	modbusReal: ModbusUnion;
END_VAR


i:= GVL.nInputRegisterIndex;

GVL.mb_Input_Registers[i+0]:= Status;

modbusReal.realValue:= Operating_Hrs;
GVL.mb_Input_Registers[i+2]:= modbusReal.wordValue[1];
GVL.mb_Input_Registers[i+3]:= modbusReal.wordValue[2];

modbusReal.realValue:= Energy;
GVL.mb_Input_Registers[i+4]:= modbusReal.wordValue[1];
GVL.mb_Input_Registers[i+5]:= modbusReal.wordValue[2];

modbusReal.realValue:= Volume;
GVL.mb_Input_Registers[i+6]:= modbusReal.wordValue[1];
GVL.mb_Input_Registers[i+7]:= modbusReal.wordValue[2];

modbusReal.realValue:= Supply_Temp;
GVL.mb_Input_Registers[i+8]:= modbusReal.wordValue[1];
GVL.mb_Input_Registers[i+9]:= modbusReal.wordValue[2];

modbusReal.realValue:= Return_Temp;
GVL.mb_Input_Registers[i+10]:= modbusReal.wordValue[1];
GVL.mb_Input_Registers[i+11]:= modbusReal.wordValue[2];

modbusReal.realValue:= Temp_Diff;
GVL.mb_Input_Registers[i+12]:= modbusReal.wordValue[1];
GVL.mb_Input_Registers[i+13]:= modbusReal.wordValue[2];

GVL.nInputRegisterIndex:= i + 14;

i:= GVL.nInputCoilIndex;

GVL.mb_Input_Coils[i+0]:= Offline;

GVL.nInputCoilIndex:= i+1;

END_FUNCTION_BLOCK

// POUs/OneFire_Suppr
FUNCTION_BLOCK OneFire_Suppr
VAR_INPUT
	Pn1_Alm : BOOL;
	Pn1_FLT: BOOL;
	Supp_Act: BOOL;
	Fire_Offline: BOOL;
END_VAR

VAR_TEMP
	i:INT;
END_VAR


i:= GVL.nInputCoilIndex;

GVL.mb_Input_Coils[i+0]:= Pn1_Alm;
GVL.mb_Input_Coils[i+1]:= Pn1_FLT;
GVL.mb_Input_Coils[i+2]:= Supp_Act;
GVL.mb_Input_Coils[i+3]:= Fire_Offline;

GVL.nInputCoilIndex:= i+4;

END_FUNCTION_BLOCK

// POUs/OneGen
FUNCTION_BLOCK OneGen
VAR_INPUT
	Run: BOOL;
	Run_Offline: BOOL;
	Warn: BOOL;
	Warn_Offline: BOOL;
	Alarm: BOOL;
	Alarm_Offline: BOOL;
	NotRdy: BOOL;
	NotRdy_Offline: BOOL;
	EmgMode: BOOL;
	EmgMode_Offline: BOOL;
END_VAR

VAR_TEMP
	i:INT;
END_VAR


i:= GVL.nInputCoilIndex;

gvl.mb_Input_Coils[i+0]:= Run;
gvl.mb_Input_Coils[i+1]:= Run_Offline;
gvl.mb_Input_Coils[i+2]:= Warn;
gvl.mb_Input_Coils[i+3]:= Warn_Offline;
gvl.mb_Input_Coils[i+4]:= Alarm;
gvl.mb_Input_Coils[i+5]:= Alarm_Offline;
gvl.mb_Input_Coils[i+6]:= NotRdy;
gvl.mb_Input_Coils[i+7]:= NotRdy_Offline;
gvl.mb_Input_Coils[i+8]:= EmgMode;
gvl.mb_Input_Coils[i+9]:= EmgMode_Offline;


GVL.nInputCoilIndex := i + 10;

END_FUNCTION_BLOCK

// POUs/OneGLP
FUNCTION_BLOCK OneGLP
VAR_INPUT
	sur_STS:BOOL;
	phs_ALM:BOOL;
	sur_phs_offline: BOOL;
	
	BRK119_POS_STS: BOOL;
	BRK119_TRIP_ALM : BOOL; 
	BRK119_offline: BOOL;
	
    BRK129_POS_STS: BOOL;
	BRK129_TRIP_ALM : BOOL; 
	BRK129_offline: BOOL;
	
    BRK450_POS_STS: BOOL;
	BRK450_TRIP_ALM : BOOL; 
	BRK450_offline: BOOL;	
END_VAR

VAR_TEMP
	i: INT;
END_VAR



i:= GVL.nInputCoilIndex;

gvl.mb_Input_Coils[i+0]:= sur_STS;
gvl.mb_Input_Coils[i+1]:= phs_ALM;
gvl.mb_Input_Coils[i+2]:= sur_phs_offline;

gvl.mb_Input_Coils[i+3]:= BRK119_POS_STS;
gvl.mb_Input_Coils[i+4]:= BRK119_TRIP_ALM;
gvl.mb_Input_Coils[i+5]:= BRK119_offline;

gvl.mb_Input_Coils[i+6]:= BRK129_POS_STS;
gvl.mb_Input_Coils[i+7]:= BRK129_TRIP_ALM;
gvl.mb_Input_Coils[i+8]:= BRK129_offline;

gvl.mb_Input_Coils[i+9]:= BRK450_POS_STS;
gvl.mb_Input_Coils[i+10]:= BRK450_TRIP_ALM;
gvl.mb_Input_Coils[i+11]:= BRK450_offline;

GVL.nInputCoilIndex:= i + 12;

END_FUNCTION_BLOCK

// POUs/OneIDF
FUNCTION_BLOCK OneIDF
VAR_INPUT
	sur_STS : BOOL;
	phs_ALM : BOOL;
	sur_phs_offline : BOOL;
	
	BRK115_POS_STS: BOOL;
	BRK115_TRIP_ALM : BOOL; 
	BRK115_offline: BOOL;
	
    BRK125_POS_STS: BOOL;
	BRK125_TRIP_ALM : BOOL; 
	BRK125_offline: BOOL;

	INCOMER_TRIP_ALM : BOOL; 
	INCOMER_offline: BOOL;
END_VAR

VAR
		i: INT;
END_VAR



i := GVL.nInputCoilIndex;

GVL.nInputCoilIndex[i+0] := sur_STS;
GVL.nInputCoilIndex[i+1] := phs_ALM;
GVL.nInputCoilIndex[i+2] := sur_phs_offline;

GVL.nInputCoilIndex[i+3] := BRK115_POS_STS;
GVL.nInputCoilIndex[i+4] := BRK115_TRIP_ALM;
GVL.nInputCoilIndex[i+5] := BRK115_offline;

GVL.nInputCoilIndex[i+6] := BRK125_POS_STS;
GVL.nInputCoilIndex[i+7] := BRK125_TRIP_ALM;
GVL.nInputCoilIndex[i+8] := BRK125_offline;

GVL.nInputCoilIndex[i+9] := INCOMER_TRIP_ALM;
GVL.nInputCoilIndex[i+10]:= INCOMER_offline;

GVL.nInputCoilIndex := i + 11;

END_FUNCTION_BLOCK

// POUs/OneIsolator_Latch
FUNCTION_BLOCK OneIsolator_Latch
VAR_INPUT
	ISO_Status: BOOL;
	OA_IsoReset: BOOL;
END_VAR
VAR_OUTPUT
	ISO_Fault: BOOL;
END_VAR
VAR
END_VAR

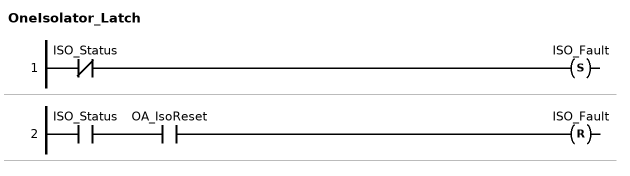
// NETWORK 1
ISO_Fault S= NOT ISO_Status;

// NETWORK 2
ISO_Fault R= ISO_Status AND OA_IsoReset;

END_FUNCTION_BLOCK

// POUs/OnePDU
FUNCTION_BLOCK OnePDU
VAR_INPUT
	sur_STS : BOOL;
	phs_ALM : BOOL;
	sur_phs_offline : BOOL;
	
	tvoc_BRK_STS: BOOL;             // CIRCUIT BREAERS
	tvoc_BRK_ALM: BOOL;            // CIRCUIT BREAERS
	tvoc_BRK_offline: BOOL; 
	
	BRK115_POS_STS: BOOL;
	BRK115_TRIP_ALM : BOOL; 
	BRK115_offline: BOOL;
	
    BRK125_POS_STS: BOOL;
	BRK125_TRIP_ALM : BOOL; 
	BRK125_offline: BOOL;
	
	BRK135_POS_STS: BOOL;
	BRK135_TRIP_ALM : BOOL; 
	BRK135_offline: BOOL;
	
    BRK215_POS_STS: BOOL;
	BRK215_TRIP_ALM : BOOL; 
	BRK215_offline: BOOL;
	
	BRK225_POS_STS: BOOL;
	BRK225_TRIP_ALM : BOOL; 
	BRK225_offline: BOOL;
	
	BRK235_POS_STS: BOOL;
	BRK235_TRIP_ALM : BOOL; 
	BRK235_offline: BOOL;
	
	BRK315_POS_STS: BOOL;
	BRK315_TRIP_ALM : BOOL; 
	BRK315_offline: BOOL;
	
    BRK325_POS_STS: BOOL;
	BRK325_TRIP_ALM : BOOL; 
	BRK325_offline: BOOL;
	
    BRK335_POS_STS: BOOL;
	BRK335_TRIP_ALM : BOOL; 
	BRK335_offline: BOOL;
	
	BRK345_POS_STS: BOOL;
	BRK345_TRIP_ALM : BOOL; 
	BRK345_offline: BOOL;

	INCOMER_RACKED_OUT : BOOL; 
	INCOMER_TRIP_ALM : BOOL; 
	INCOMER_offline: BOOL;

END_VAR

VAR_TEMP
	i: INT;
END_VAR


i := GVL.nInputCoilIndex;
GVL.mb_Input_Coils[i+0] := sur_STS;
GVL.mb_Input_Coils[i+1] := phs_ALM;
GVL.mb_Input_Coils[i+2] := sur_phs_offline;

GVL.mb_Input_Coils[i+3] := tvoc_BRK_STS ;
GVL.mb_Input_Coils[i+4] := tvoc_BRK_ALM ;
GVL.mb_Input_Coils[i+5] := tvoc_BRK_offline;

GVL.mb_Input_Coils[i+6] := BRK115_POS_STS;
GVL.mb_Input_Coils[i+7] := BRK115_TRIP_ALM;
GVL.mb_Input_Coils[i+8] := BRK115_offline;

GVL.mb_Input_Coils[i+9] := BRK125_POS_STS;
GVL.mb_Input_Coils[i+10] := BRK125_TRIP_ALM;
GVL.mb_Input_Coils[i+11] := BRK125_offline;

GVL.mb_Input_Coils[i+12] := BRK135_POS_STS;
GVL.mb_Input_Coils[i+13] := BRK135_TRIP_ALM;
GVL.mb_Input_Coils[i+14] := BRK135_offline;

GVL.mb_Input_Coils[i+15] := BRK215_POS_STS;
GVL.mb_Input_Coils[i+16] := BRK215_TRIP_ALM;
GVL.mb_Input_Coils[i+17] := BRK215_offline;

GVL.mb_Input_Coils[i+18] := BRK225_POS_STS;
GVL.mb_Input_Coils[i+19] := BRK225_TRIP_ALM;
GVL.mb_Input_Coils[i+20] := BRK225_offline;

GVL.mb_Input_Coils[i+21] := BRK235_POS_STS;
GVL.mb_Input_Coils[i+22] := BRK235_TRIP_ALM;
GVL.mb_Input_Coils[i+23] := BRK235_offline;

GVL.mb_Input_Coils[i+24] := BRK315_POS_STS;
GVL.mb_Input_Coils[i+25] := BRK315_TRIP_ALM;
GVL.mb_Input_Coils[i+26] := BRK315_offline;

GVL.mb_Input_Coils[i+27] := BRK325_POS_STS;
GVL.mb_Input_Coils[i+28] := BRK325_TRIP_ALM;
GVL.mb_Input_Coils[i+29] := BRK325_offline;

GVL.mb_Input_Coils[i+30] := BRK335_POS_STS;
GVL.mb_Input_Coils[i+31] := BRK335_TRIP_ALM;
GVL.mb_Input_Coils[i+32] := BRK335_Offline;

GVL.mb_Input_Coils[i+33] := BRK345_POS_STS;
GVL.mb_Input_Coils[i+34] := BRK345_TRIP_ALM;
GVL.mb_Input_Coils[i+35] := BRK345_Offline;

GVL.mb_Input_Coils[i+36] := INCOMER_RACKED_OUT;
GVL.mb_Input_Coils[i+37] := INCOMER_TRIP_ALM;
GVL.mb_Input_Coils[i+38] := INCOMER_offline;

GVL.nInputCoilIndex := i + 39;

END_FUNCTION_BLOCK

// POUs/OnePumpFF_Latch
FUNCTION_BLOCK OnePumpFF_Latch
VAR_INPUT
	DP_Switch: BOOL;
	Pump_Run: BOOL;
	OA_AlarmReset: BOOL;
	PumpFailureDelay: TIME;
END_VAR
VAR_OUTPUT
	PumpFlow_Alarm: BOOL;
END_VAR
VAR
	NoFlow: BOOL;
	T1: TON;
END_VAR

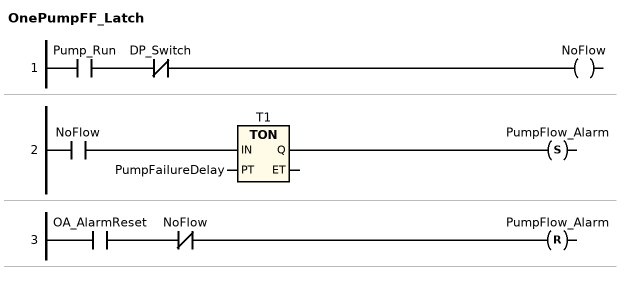
// NETWORK 1
NoFlow := Pump_Run AND NOT DP_Switch;

// NETWORK 2
T1(IN := NoFlow, PT := PumpFailureDelay); // TON
PumpFlow_Alarm S= T1.Q;

// NETWORK 3
PumpFlow_Alarm R= OA_AlarmReset AND NOT NoFlow;

END_FUNCTION_BLOCK

// POUs/OneSpeed_Override
FUNCTION_BLOCK OneSpeed_Override
VAR_INPUT
	Master_Speed : REAL;
	Pump_Ovr: BOOL;
	OA_Speed: REAL;
	OA_SpeedMin: REAL;
	OA_SpeedMax: REAL;
	
END_VAR
VAR_OUTPUT
	VSD_Speed: REAL;
	
END_VAR
VAR
END_VAR

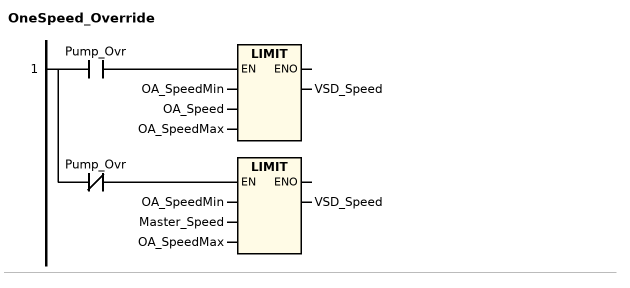
// NETWORK 1
IF Pump_Ovr THEN VSD_Speed := LIMIT(OA_SpeedMin, OA_Speed, OA_SpeedMax); END_IF
IF NOT Pump_Ovr THEN VSD_Speed := LIMIT(OA_SpeedMin, Master_Speed, OA_SpeedMax); END_IF

END_FUNCTION_BLOCK

// POUs/OneSTS
FUNCTION_BLOCK OneSTS
VAR_INPUT
	Trans_Inhibt : BOOL;
	Trans_Inhibt_Offline : BOOL;
    Com_Alm : BOOL;
	Com_Alm_Offline: BOOL;
    Fan_Fail : BOOL;
	Fan_Fail_Offline : BOOL;
	
    Load_Line_1 : BOOL;
	Load_Line_1_Offline : BOOL;
    Load_Line_2 : BOOL;
	Load_Line_2_Offline : BOOL;
	
    Load_Line_1_ByPass : BOOL;
	LL_1_ByPass_offline : BOOL;
    Load_Line_2_ByPass : BOOL;
	LL_2_ByPass_offline : BOOL;
	Load_DisCon : BOOL;
	Load_DisCon_Offline : BOOL;
END_VAR

VAR_OUTPUT
	STS_Inhibited : BOOL;
END_VAR

VAR_TEMP
	i:INT;
END_VAR



i:= GVL.nInputCoilIndex;

GVL.mb_Input_Coils[i+0]:= Trans_Inhibt;
GVL.mb_Input_Coils[i+1]:= Trans_Inhibt_Offline;

GVL.mb_Input_Coils[i+2]:= Com_Alm;
GVL.mb_Input_Coils[i+3]:= Com_Alm_Offline;

GVL.mb_Input_Coils[i+4]:= Fan_Fail;
GVL.mb_Input_Coils[i+5]:= Fan_Fail_Offline;

GVL.mb_Input_Coils[i+6]:= Load_Line_1;
GVL.mb_Input_Coils[i+7]:= Load_Line_1_Offline;

GVL.mb_Input_Coils[i+8]:= Load_Line_2;
GVL.mb_Input_Coils[i+9]:= Load_Line_2_Offline;

GVL.mb_Input_Coils[i+10]:= Load_Line_1_ByPass;
GVL.mb_Input_Coils[i+11]:= LL_1_ByPass_offline;

GVL.mb_Input_Coils[i+12]:= Load_Line_2_ByPass;
GVL.mb_Input_Coils[i+13]:= LL_2_ByPass_offline;

GVL.mb_Input_Coils[i+14]:= Load_DisCon;
GVL.mb_Input_Coils[i+15]:= Load_DisCon_Offline;

GVL.nInputCoilIndex:= i+16; 

i:= GVL.nOutputCoilIndex;
STS_Inhibited:= GVL.mb_Output_Coils[i+0];

GVL.nOutputCoilIndex:= i + 1;

END_FUNCTION_BLOCK

// POUs/OneSTS_RTU
FUNCTION_BLOCK OneSTS_RTU
VAR_INPUT
	STS_Num: INT;
END_VAR

VAR_TEMP
	i:INT;
	modbusReal: ModbusUnion;
END_VAR


i:=GVL.nInputRegisterIndex;

modbusReal.realValue:= GVL_STS.STS[STS_Num].PRI_VA;
GVL.mb_Input_Registers[i+0] := modbusReal.wordValue[1];
GVL.mb_Input_Registers[i+1] := modbusReal.wordValue[2];


modbusReal.realValue:= GVL_STS.STS[STS_Num].PRI_VB;
GVL.mb_Input_Registers[i+2] := modbusReal.wordValue[1];
GVL.mb_Input_Registers[i+3] := modbusReal.wordValue[2];

modbusReal.realValue:= GVL_STS.STS[STS_Num].PRI_VC;
GVL.mb_Input_Registers[i+4] := modbusReal.wordValue[1];
GVL.mb_Input_Registers[i+5] := modbusReal.wordValue[2];

modbusReal.realValue:= GVL_STS.STS[STS_Num].OTP_VA;
GVL.mb_Input_Registers[i+6] := modbusReal.wordValue[1];
GVL.mb_Input_Registers[i+7] := modbusReal.wordValue[2];

modbusReal.realValue:= GVL_STS.STS[STS_Num].OTP_VB;
GVL.mb_Input_Registers[i+8] := modbusReal.wordValue[1];
GVL.mb_Input_Registers[i+9] := modbusReal.wordValue[2];

modbusReal.realValue:= GVL_STS.STS[STS_Num].OTP_VC;
GVL.mb_Input_Registers[i+10] := modbusReal.wordValue[1];
GVL.mb_Input_Registers[i+11] := modbusReal.wordValue[2];


modbusReal.realValue:= GVL_STS.STS[STS_Num].AMPSA;
GVL.mb_Input_Registers[i+12] := modbusReal.wordValue[1];
GVL.mb_Input_Registers[i+13] := modbusReal.wordValue[2];

modbusReal.realValue:= GVL_STS.STS[STS_Num].AMPSB;
GVL.mb_Input_Registers[i+14] := modbusReal.wordValue[1];
GVL.mb_Input_Registers[i+15] := modbusReal.wordValue[2];


modbusReal.realValue:= GVL_STS.STS[STS_Num].AMPSC;
GVL.mb_Input_Registers[i+16] := modbusReal.wordValue[1];
GVL.mb_Input_Registers[i+17] := modbusReal.wordValue[2];

modbusReal.realValue:= GVL_STS.STS[STS_Num].FREQ;
GVL.mb_Input_Registers[i+18] := modbusReal.wordValue[1];
GVL.mb_Input_Registers[i+19] := modbusReal.wordValue[2];

modbusReal.realValue:= GVL_STS.STS[STS_Num].SEC_VA;
GVL.mb_Input_Registers[i+20] := modbusReal.wordValue[1];
GVL.mb_Input_Registers[i+21] := modbusReal.wordValue[2];

modbusReal.realValue:= GVL_STS.STS[STS_Num].SEC_VB;
GVL.mb_Input_Registers[i+22] := modbusReal.wordValue[1];
GVL.mb_Input_Registers[i+23] := modbusReal.wordValue[2];

modbusReal.realValue:= GVL_STS.STS[STS_Num].SEC_VC;
GVL.mb_Input_Registers[i+24] := modbusReal.wordValue[1];
GVL.mb_Input_Registers[i+25] := modbusReal.wordValue[2];

modbusReal.realValue:= GVL_STS.STS[STS_Num].OTP_LOAD_A;
GVL.mb_Input_Registers[i+26] := modbusReal.wordValue[1];
GVL.mb_Input_Registers[i+27] := modbusReal.wordValue[2];

modbusReal.realValue:= GVL_STS.STS[STS_Num].OTP_LOAD_B;
GVL.mb_Input_Registers[i+28] := modbusReal.wordValue[1];
GVL.mb_Input_Registers[i+29] := modbusReal.wordValue[2];

modbusReal.realValue:= GVL_STS.STS[STS_Num].OTP_LOAD_C;
GVL.mb_Input_Registers[i+30] := modbusReal.wordValue[1];
GVL.mb_Input_Registers[i+31] := modbusReal.wordValue[2];

modbusReal.realValue:= GVL_STS.STS[STS_Num].OTP_KW_A;
GVL.mb_Input_Registers[i+32] := modbusReal.wordValue[1];
GVL.mb_Input_Registers[i+33] := modbusReal.wordValue[2];

modbusReal.realValue:= GVL_STS.STS[STS_Num].OTP_KW_B;
GVL.mb_Input_Registers[i+34] := modbusReal.wordValue[1];
GVL.mb_Input_Registers[i+35] := modbusReal.wordValue[2];

modbusReal.realValue:= GVL_STS.STS[STS_Num].OTP_KW_C;
GVL.mb_Input_Registers[i+36] := modbusReal.wordValue[1];
GVL.mb_Input_Registers[i+37] := modbusReal.wordValue[2];

modbusReal.realValue:= GVL_STS.STS[STS_Num].OTP_KVA_A;
GVL.mb_Input_Registers[i+38] := modbusReal.wordValue[1];
GVL.mb_Input_Registers[i+39] := modbusReal.wordValue[2];

modbusReal.realValue:= GVL_STS.STS[STS_Num].OTP_KVA_B;
GVL.mb_Input_Registers[i+40] := modbusReal.wordValue[1];
GVL.mb_Input_Registers[i+41] := modbusReal.wordValue[2];

modbusReal.realValue:= GVL_STS.STS[STS_Num].OTP_KVA_C;
GVL.mb_Input_Registers[i+42] := modbusReal.wordValue[1];
GVL.mb_Input_Registers[i+43] := modbusReal.wordValue[2];

modbusReal.realValue:= GVL_STS.STS[STS_Num].PF_A;
GVL.mb_Input_Registers[i+44] := modbusReal.wordValue[1];
GVL.mb_Input_Registers[i+45] := modbusReal.wordValue[2];

modbusReal.realValue:= GVL_STS.STS[STS_Num].PF_B;
GVL.mb_Input_Registers[i+46] := modbusReal.wordValue[1];
GVL.mb_Input_Registers[i+47] := modbusReal.wordValue[2];

modbusReal.realValue:= GVL_STS.STS[STS_Num].PF_C;
GVL.mb_Input_Registers[i+48] := modbusReal.wordValue[1];
GVL.mb_Input_Registers[i+49] := modbusReal.wordValue[2];

GVL.nInputRegisterIndex:= i + 50;

i:=GVL.nInputCoilIndex;

GVL.mb_Input_Coils[i+0] := GVL_STS.STS[STS_Num].COM_ALM;
GVL.mb_Input_Coils[i+1] := GVL_STS.STS[STS_Num].OTP_BKR_OPN;
GVL.mb_Input_Coils[i+2] := GVL_STS.STS[STS_Num].L1_INP_BKR_OPN;
GVL.mb_Input_Coils[i+3] := GVL_STS.STS[STS_Num].L2_INP_BKR_OPN;
GVL.mb_Input_Coils[i+4] := GVL_STS.STS[STS_Num].L1_BYP_BKR_TRP;
GVL.mb_Input_Coils[i+5] := GVL_STS.STS[STS_Num].L2_BYP_BKR_TRP;
GVL.mb_Input_Coils[i+6] := GVL_STS.STS[STS_Num].OTP_BKR_TRP;
GVL.mb_Input_Coils[i+7] := GVL_STS.STS[STS_Num].L1_INP_BKR_TRP;
GVL.mb_Input_Coils[i+8] := GVL_STS.STS[STS_Num].L2_INP_BKR_TRP;
GVL.mb_Input_Coils[i+9] := GVL_STS.STS[STS_Num].FANS_FAIL;

GVL.nInputRegisterIndex:= i + 10;

END_FUNCTION_BLOCK

// POUs/OneSWBL
FUNCTION_BLOCK OneSWBL
VAR_INPUT
	sur_STS : BOOL;
	phs_ALM_1 : BOOL;
	phs_ALM_2 : BOOL;
	sur_phs_offline : BOOL;
	
	Etherm_24VDC_STS : BOOL;
	Etherm_24VDC_Offline: BOOL;
	
	tvoc_BRK_STS: BOOL;               // CIRCUIT BREAERS
	tvoc_BRK_ALM: BOOL; 
    tvoc_24VDC_STS : BOOL;           // CIRCUIT BREAERS
	tvoc_BRK_offline: BOOL; 
	
	BRK_FC11_POS_STS: BOOL;
	BRK_FC11_TRIP_ALM : BOOL; 
	BRK_FC11_offline: BOOL;
	
	BRK_BA01_POS_STS: BOOL;
	BRK_BA01_TRIP_ALM : BOOL; 
	BRK_BA01_offline: BOOL;
	
    BRK_EC01_POS_STS: BOOL;
	BRK_EC01_TRIP_ALM : BOOL; 
	BRK_EC01_offline: BOOL;
	
	BRK_JA01_POS_STS: BOOL;
	BRK_JA01_TRIP_ALM : BOOL; 
	BRK_JA01_offline: BOOL;
	
    BRK_MC01_POS_STS: BOOL;
	BRK_MC01_TRIP_ALM : BOOL; 
	BRK_MC01_offline: BOOL;
	
	BRK_RA01_POS_STS: BOOL;
	BRK_RA01_TRIP_ALM : BOOL; 
	BRK_RA01_offline: BOOL;
	
	
	BRK_NO2_BA01_POS_STS: BOOL;
	BRK_NO2_BA01_TRIP_ALM : BOOL; 
	BRK_NO2_BA01_offline: BOOL;
END_VAR

VAR_TEMP
	i:INT;
END_VAR


i := GVL.nInputCoilIndex;

GVL.mb_Input_Coils[i+0] := sur_STS;
GVL.mb_Input_Coils[i+1] := phs_ALM_1;
GVL.mb_Input_Coils[i+2] := phs_ALM_2;
GVL.mb_Input_Coils[i+3] := sur_phs_offline;

GVL.mb_Input_Coils[i+4] := sur_STS;
GVL.mb_Input_Coils[i+5] := phs_ALM_1;

GVL.mb_Input_Coils[i+6] := tvoc_BRK_STS;
GVL.mb_Input_Coils[i+7] := tvoc_BRK_ALM;
GVL.mb_Input_Coils[i+8] := tvoc_24VDC_STS;
GVL.mb_Input_Coils[i+9] := tvoc_BRK_offline;

GVL.mb_Input_Coils[i+10] := BRK_FC11_POS_STS;
GVL.mb_Input_Coils[i+11] := BRK_FC11_TRIP_ALM;
GVL.mb_Input_Coils[i+12] := BRK_FC11_offline;

GVL.mb_Input_Coils[i+13] := BRK_BA01_POS_STS;
GVL.mb_Input_Coils[i+14] := BRK_BA01_TRIP_ALM;
GVL.mb_Input_Coils[i+15] := BRK_BA01_offline;

GVL.mb_Input_Coils[i+16] := BRK_EC01_POS_STS;
GVL.mb_Input_Coils[i+17] := BRK_EC01_TRIP_ALM;
GVL.mb_Input_Coils[i+18] := BRK_EC01_offline;

GVL.mb_Input_Coils[i+19] := BRK_JA01_POS_STS;
GVL.mb_Input_Coils[i+20] := BRK_JA01_TRIP_ALM;
GVL.mb_Input_Coils[i+21] := BRK_JA01_offline;

GVL.mb_Input_Coils[i+22] := BRK_MC01_POS_STS;
GVL.mb_Input_Coils[i+23] := BRK_MC01_TRIP_ALM;
GVL.mb_Input_Coils[i+24] := BRK_MC01_offline;

GVL.mb_Input_Coils[i+25] := BRK_RA01_POS_STS;
GVL.mb_Input_Coils[i+26] := BRK_RA01_TRIP_ALM;
GVL.mb_Input_Coils[i+27] := BRK_RA01_offline;

GVL.mb_Input_Coils[i+28] := BRK_NO2_BA01_POS_STS;
GVL.mb_Input_Coils[i+29] := BRK_NO2_BA01_TRIP_ALM;
GVL.mb_Input_Coils[i+30] := BRK_NO2_BA01_offline;


GVL.nInputCoilIndex := i + 31;

END_FUNCTION_BLOCK

// POUs/OneTie_BRK
FUNCTION_BLOCK OneTie_BRK
VAR_INPUT
	
	TIEBKR_STS: BOOL;
	TIEBKR_STS_Offline: BOOL;
	
	TIEBKR_RCKIN : BOOL;
	TIEBKR_RCKIN_Offline : BOOL;
	
	TIEBKR_TEST : BOOL;
	TIEBKR_TEST_Offline : BOOL;
	
	TIEBKR_RCKOUT : BOOL;
	TIEBKR_RCKOUT_Offline : BOOL;

END_VAR

VAR_TEMP
	i:INT;
END_VAR


i:= GVL.nInputCoilIndex;

GVL.mb_Input_Coils[i+0] := TIEBKR_STS;
GVL.mb_Input_Coils[i+1] := TIEBKR_STS_Offline;

GVL.mb_Input_Coils[i+2] := TIEBKR_RCKIN;
GVL.mb_Input_Coils[i+3] := TIEBKR_RCKIN_Offline;

GVL.mb_Input_Coils[i+4] := TIEBKR_TEST;
GVL.mb_Input_Coils[i+5] := TIEBKR_TEST_Offline;

GVL.mb_Input_Coils[i+6] := TIEBKR_RCKOUT;
GVL.mb_Input_Coils[i+7] := TIEBKR_RCKOUT_Offline;

GVL.nInputCoilIndex := i + 8;

END_FUNCTION_BLOCK

// POUs/OneUPS
FUNCTION_BLOCK OneUPS
VAR_INPUT
	Crit_Alm : BOOL;
	Minor_Alm : BOOL;
	ByPass_Mode : BOOL;
	Batt_Mode : BOOL;
	Offline: BOOL;
END_VAR

VAR_TEMP
	i : INT;
END_VAR

i:= GVL.nInputCoilIndex;

GVL.mb_Input_Coils[i+0] := Crit_Alm;
GVL.mb_Input_Coils[i+1] := Minor_Alm;
GVL.mb_Input_Coils[i+2] := ByPass_Mode;
GVL.mb_Input_Coils[i+3] := Batt_Mode;
GVL.mb_Input_Coils[i+4] := Offline;

GVL.nInputCoilIndex := i + 5;

END_FUNCTION_BLOCK

// POUs/OneVSD_Latch
FUNCTION_BLOCK OneVSD_Latch
VAR_INPUT
	VSD_Run: BOOL;
	VSD_Fault: BOOL;
	VSD_Delay: TIME;
	OA_VSDReset: BOOL;
	
END_VAR
VAR_OUTPUT
	VSD_FaultAct: BOOL;
END_VAR
VAR
	T1:TON;
END_VAR

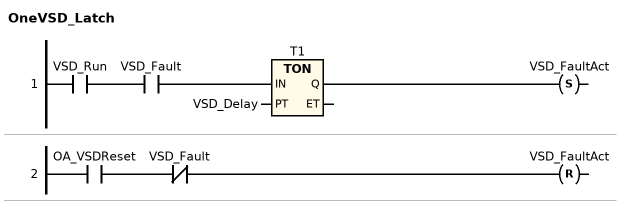
// NETWORK 1
T1(IN := VSD_Run AND VSD_Fault, PT := VSD_Delay); // TON
VSD_FaultAct S= T1.Q;

// NETWORK 2
VSD_FaultAct R= OA_VSDReset AND NOT VSD_Fault;

END_FUNCTION_BLOCK

// POUs/ReadModbusBool
FUNCTION ReadModbusBool : bool
VAR_INPUT
END_VAR
VAR
	i: INT;
	modbusBool: BOOL;
END_VAR

i := GVL.nOutputCoilIndex;

modbusBool := GVL.mb_Output_Coils[i+0];

GVL.nOutputCoilIndex := i+1;

ReadModbusBool:= modbusBool;

END_FUNCTION

// POUs/ReadModbusReal
FUNCTION ReadModbusReal : REAL
VAR
	i: INT;
	modbusReal: ModbusUnion;
END_VAR


i:= GVL.nOutputRegisterIndex;

modbusReal.wordValue[1]:= GVL.mb_Output_Registers[i+0];
modbusReal.wordValue[2]:= GVL.mb_Output_Registers[i+1];

GVL.nOutputRegisterIndex:= i + 2;

ReadModbusReal:=modbusReal.realValue;

END_FUNCTION

// POUs/ReadModusTime
FUNCTION ReadModusTime : Time
VAR_INPUT
END_VAR
VAR
	i: INT;
	modbusTime: ModbusUnion;
END_VAR


i:= GVL.nOutputRegisterIndex;

modbusTime.longValue:= GVL.mb_Output_Registers[i+0] * 1000;

GVL.nOutputRegisterIndex:= i + 0;


ReadModusTime := modbusTime.timeValue;

END_FUNCTION

// POUs/WriteModbusBool
FUNCTION_BLOCK WriteModbusBool
VAR_INPUT
	L_Input: BOOL;
END_VAR
VAR_OUTPUT
END_VAR
VAR
	i: INT;
END_VAR


i:= GVL.nInputCoilIndex;
GVL.mb_Input_Coils[i+0]:= L_Input;

GVL.nInputCoilIndex:= i+1;

END_FUNCTION_BLOCK

// POUs/WriteModbusReal
FUNCTION_BLOCK WriteModbusReal
VAR_INPUT
	L_input: REAL;	
END_VAR
VAR
	i: INT;
	modbusReal: ModbusUnion;
END_VAR


i:= GVL.nInputRegisterIndex;
modbusReal.realValue:= L_input;

GVL.nInputRegisterIndex[i+0]:= modbusReal.wordValue[1];
GVL.nInputRegisterIndex[i+1]:= modbusReal.wordValue[2];
GVL.nInputRegisterIndex:= i+2;

END_FUNCTION_BLOCK

// POUs/WriteModbusWord
FUNCTION_BLOCK WriteModbusWord
VAR_INPUT
	L_input: WORD;
END_VAR
VAR_OUTPUT
END_VAR
VAR
	i: INT;
END_VAR


i:= GVL.nInputRegisterIndex;

GVL.mb_Input_Registers[i+0]:= L_input;
GVL.nInputRegisterIndex:= i+1;

END_FUNCTION_BLOCK

// VISUs/AminCRAH
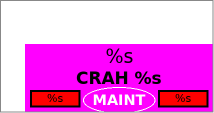
VISUALIZATION AminCRAH  // 214x113
VAR_INPUT
	idCrah : WSTRING;
	Offline : BOOL;
	Alarm : BOOL;
	Enable: BOOL;
	Running: BOOL;
	Inhibited : BOOL;
	Maintenance : BOOL;		
	HOA : WORD;
	Isolator1 : BOOL;
	Isolator2 : BOOL;
	DeactivateIso2 : BOOL;
END_VAR
    Rectangle (24,43 190x70), colour toggle: Enable
    Rectangle (24,43 190x70), colour toggle: Enable, invisible if: Not Running
    Rectangle (24,43 190x70), colour toggle: Enable, invisible if: Not Inhibited
    Rectangle (24,43 190x70), colour toggle: Enable, invisible if: Not Offline
    Rectangle (24,43 190x70), "CRAH %s", text variable: idCrah, colour toggle: Enable, invisible if: Not Inhibited
    Rectangle (84,46 71x21), "%s", text list: 'CRAH_Status', text index: HOA
    Ellipse (83,87 72x26), "MAINT", invisible if: Not Inhibited
    Rectangle (30,90 50x17), "%s", colour toggle: Isolator1, text list: 'CRAH_Isolator_Status', text index: Isolator1
    Rectangle (158,90 50x17), "%s", colour toggle: Isolator2, text list: 'CRAH_Isolator_Status', text index: Isolator2
END_VISUALIZATION

// VISUs/Dialog_CRAH
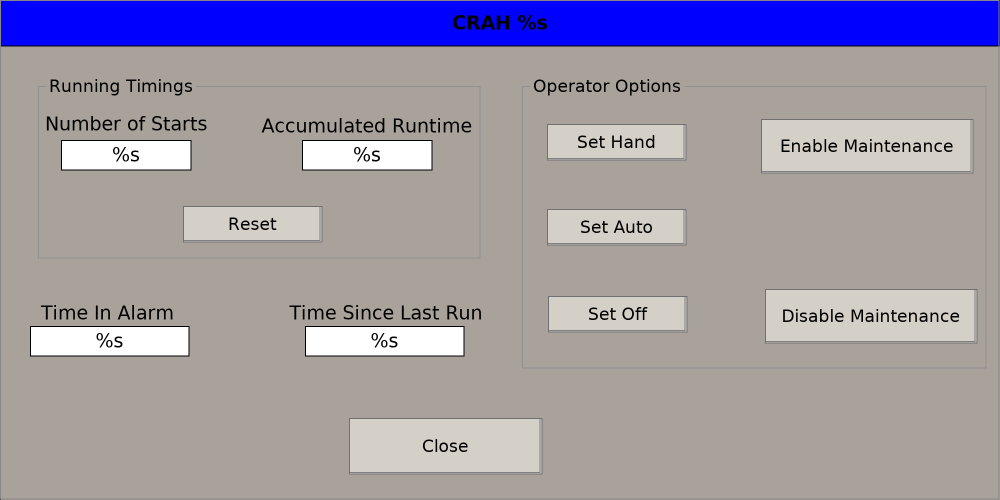
VISUALIZATION Dialog_CRAH  // 1000x500
VAR_IN_OUT
	sHeader : WSTRING;
	bCommonAlarm : BOOL;
	bIsolator1Alm :BOOL;
	bIsolator2Alm :BOOL;
	nSetControl :WORD;
	iNumStarts : WORD;
	sAccTime : STRING;
	sAlarmTime : STRING;
	sLastRunTime : STRING;
	bSetMaintenance : BOOL;
	bResetTimings : BOOL;
END_VAR
    GroupBox (38,78 442x180), "Running Timings"
        Button (145,128 139x36), "Reset"
            OnMouseClick: execute { bResetTimings:=1; }
    Rectangle (0,0 1000x46), "CRAH %s", text variable: sHeader
    Label (29,298 157x30), "Time In Alarm"
    Rectangle (30,326 159x30), "%s", text variable: sAlarmTime
    Label (39,109 175x30), "Number of Starts"
    Rectangle (61,140 130x30), "%s", text variable: iNumStarts
    Label (257,111 220x30), "Accumulated Runtime"
    Rectangle (302,140 130x30), "%s", text variable: sAccTime
    Label (285,298 202x30), "Time Since Last Run"
    Rectangle (305,326 159x30), "%s", text variable: sLastRunTime
    GroupBox (522,78 464x290), "Operator Options"
        Button (25,46 139x36), "Set Hand"
            OnMouseClick: execute { nSetControl:= 0; }
            OnMouseClick:  Dialog=Dialog_CRAH, Result=OK, NumpadKeypadSet=True
        Button (25,131 139x36), "Set Auto"
            OnMouseClick: execute { nSetControl:= 2; }
            OnMouseClick:  Dialog=Dialog_CRAH, Result=OK, NumpadKeypadSet=True
        Button (26,218 139x36), "Set Off"
            OnMouseClick: execute { nSetControl:= 1; }
            OnMouseClick:  Dialog=Dialog_CRAH, Result=OK, NumpadKeypadSet=True
        Button (239,41 212x54), "Enable Maintenance"
            OnMouseClick: execute { bSetMaintenance:= 1; }
            OnMouseClick:  Dialog=Dialog_CRAH, Result=OK, NumpadKeypadSet=True
        Button (243,211 212x54), "Disable Maintenance"
            OnMouseClick: execute { bSetMaintenance:= 0; }
            OnMouseClick:  Dialog=Dialog_CRAH, Result=OK, NumpadKeypadSet=True
    Button (349,418 193x56), "Close"
        OnMouseClick:  Dialog=Dialog_CRAH, Result=OK, NumpadKeypadSet=True
    Line (1000,0) (1000,500)
    Line (0,0) (0,500)
    Line (0,500) (1000,500)
END_VISUALIZATION

// VISUs/Dialog_DP_Field
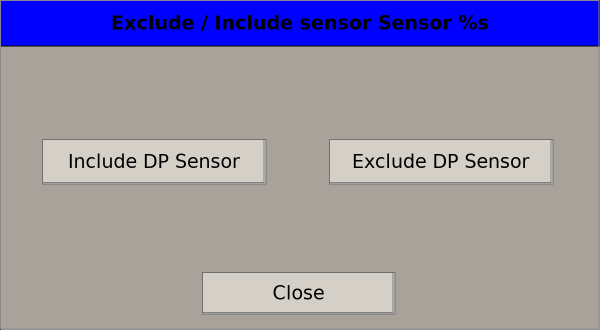
VISUALIZATION Dialog_DP_Field  // 600x330
VAR_IN_OUT
	sHeader: STRING;
	bSetPressIncluded: BOOL;
	bSetPressExcluded: BOOL;

END_VAR
    Rectangle (0,0 600x46), "Exclude / Include sensor Sensor %s", text variable: sHeader
    Button (42,139 224x45), "Include DP Sensor"
        OnMouseClick: execute { bSetPressIncluded:= TRUE; }
        OnMouseClick:  Dialog=Dialog_CRAH, Result=OK, NumpadKeypadSet=True
    Button (329,139 224x45), "Exclude DP Sensor"
        OnMouseClick: execute { bSetPressExcluded:= TRUE; }
        OnMouseClick:  Dialog=Dialog_DP_Field, Result=OK, NumpadKeypadSet=True
    Button (202,272 193x42), "Close"
        OnMouseClick: execute { bSetPressIncluded:= TRUE; }
        OnMouseClick:  Dialog=Dialog_CRAH, Result=OK, NumpadKeypadSet=True
    Line (600,0) (600,330)
    Line (0,0) (0,330)
    Line (0,330) (600,330)
    Line (0,0) (600,0)
END_VISUALIZATION

// VISUs/Dialog_EnergyMeter
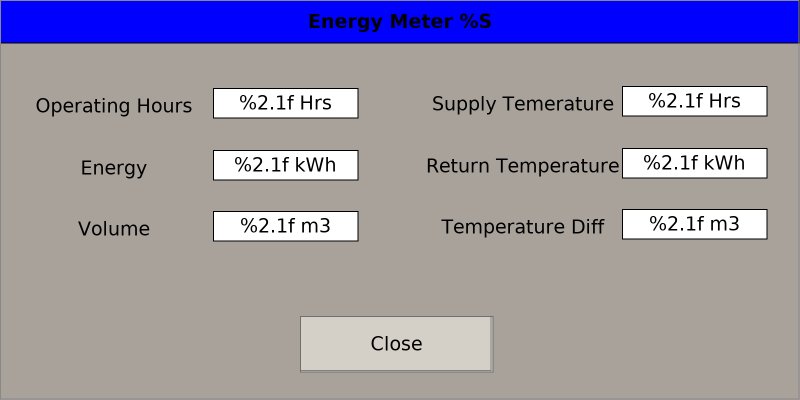
VISUALIZATION Dialog_EnergyMeter  // 800x400
VAR_IN_OUT
	sHeader : STRING;
	fOperHours: REAL;
	fEnergy: REAL;
	fVolume: REAL;
	fSupply_Temp:REAL;
	fReturn_Temp : REAL;
	fReturn_Diff: REAL;

END_VAR
    Rectangle (0,0 800x43), "Energy Meter %S", text variable: sHeader
    Label (19,92 190x28), "Operating Hours"
    Label (19,154 190x28), "Energy"
    Label (19,215 190x28), "Volume"
    Rectangle (213,88 145x30), "%2.1f Hrs", text variable: fOperHours
    Rectangle (213,150 145x30), "%2.1f kWh", text variable: fEnergy
    Rectangle (213,211 145x30), "%2.1f m3", text variable: fVolume
    Label (428,90 190x28), "Supply Temerature"
    Label (428,152 190x28), "Return Temperature"
    Label (428,213 190x28), "Temperature Diff"
    Rectangle (622,86 145x30), "%2.1f Hrs", text variable: fSupply_Temp
    Rectangle (622,148 145x30), "%2.1f kWh", text variable: fReturn_Temp
    Rectangle (622,209 145x30), "%2.1f m3", text variable: fReturn_Diff
    Button (300,316 193x56), "Close"
END_VISUALIZATION

// VISUs/Dialog_PDU
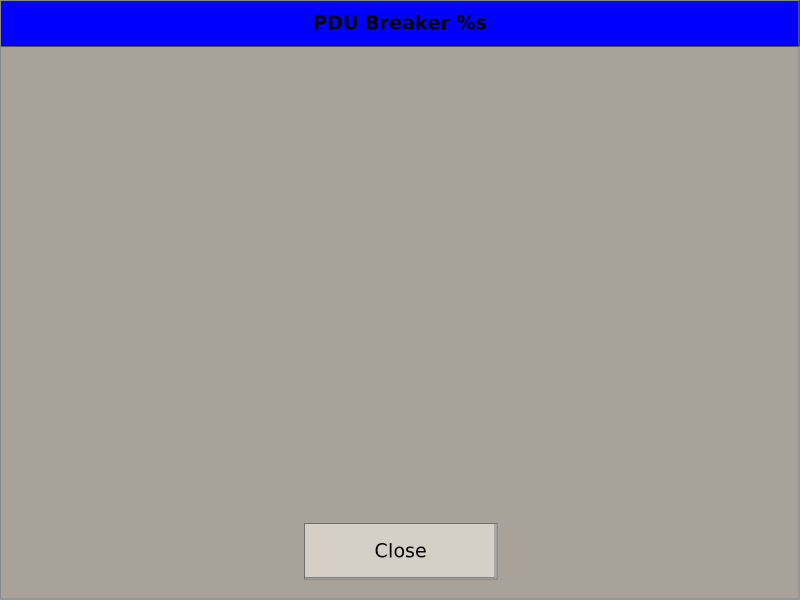
VISUALIZATION Dialog_PDU  // 800x600
VAR_IN_OUT
	sHeader : WSTRING;
	bCommonAlarm : BOOL;
	bIsolator1Alm :BOOL;
	bIsolator2Alm :BOOL;
END_VAR
    Rectangle (0,0 800x46), "PDU Breaker %s", text variable: sHeader
    Button (304,523 193x56), "Close"
        OnMouseClick:  Dialog=Dialog_CRAH, Result=OK, NumpadKeypadSet=True
END_VISUALIZATION

// VISUs/Dialog_THT_Field
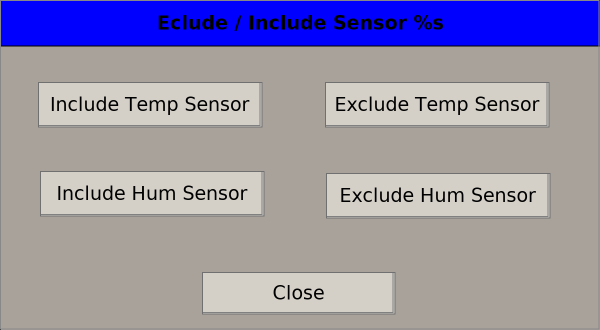
VISUALIZATION Dialog_THT_Field  // 600x330
VAR_IN_OUT
	sHeader : STRING;
	bSetTempIncluded : BOOL;
	bSetHumIncluded : BOOL;
	bSetTempExcluded : BOOL;
	bSetHumExcluded : BOOL;
END_VAR
    Rectangle (0,0 601x46), "Eclude / Include Sensor %s", text variable: sHeader
    Button (38,82 224x45), "Include Temp Sensor"
        OnMouseClick: execute { bSetTempIncluded:= TRUE; }
        OnMouseClick:  Dialog=Dialog_CRAH, Result=OK, NumpadKeypadSet=True
    Button (40,171 224x45), "Include Hum Sensor"
        OnMouseClick: execute { bSetHumIncluded:= TRUE; }
        OnMouseClick:  Dialog=Dialog_CRAH, Result=OK, NumpadKeypadSet=True
    Button (325,82 224x45), "Exclude Temp Sensor"
        OnMouseClick: execute { bSetTempExcluded:= TRUE; }
        OnMouseClick:  Dialog=Dialog_CRAH, Result=OK, NumpadKeypadSet=True
    Button (326,173 224x45), "Exclude Hum Sensor"
        OnMouseClick: execute { bSetHumExcluded:= TRUE; }
        OnMouseClick:  Dialog=Dialog_CRAH, Result=OK, NumpadKeypadSet=True
    Button (202,272 193x42), "Close"
        OnMouseClick:  Dialog=Dialog_CRAH, Result=OK, NumpadKeypadSet=True
    Line (600,0) (600,330)
    Line (0,330) (600,330)
    Line (0,0) (0,330)
    Line (0,0) (600,0)
END_VISUALIZATION

// VISUs/Obj_Alarm_Equipment
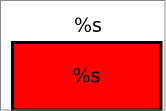
VISUALIZATION Obj_Alarm_Equipment  // 166x111
VAR_INPUT
	sIndex : STRING;
	bAlarm : BOOL;
	bOffline : BOOL;
END_VAR
    Rectangle (11,41 151x70), "%s", invisible if: bOffline
    Rectangle (10,7 156x37), "%s", text variable: sIndex
    Rectangle (11,41 151x70), "%s", colour toggle: bAlarm
END_VISUALIZATION

// VISUs/Obj_DP_Field
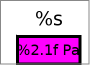
VISUALIZATION Obj_DP_Field  // 90x65
VAR_IN
	rPressValue : REAL;
	sIndex : STRING;
	bPressLimitAlarm : BOOL;
	bPressFailed : BOOL;
	bPressOffline : BOOL;
	bPressExcluded : BOOL;
END_VAR

VAR_IN_OUT
	bSetPressExcluded : BOOL;
	bSetPressIncluded : BOOL;
END_VAR
    Rectangle (16,35 65x30), "%2.1f Pa", text variable: rPressValue, colour toggle: bPressLimitAlarm
    Rectangle (8,4 82x30), "%s", text variable: sIndex
    Rectangle (16,35 65x30), "%2.1f Pa", text variable: rPressValue, invisible if: not bPressExcluded
    Rectangle (16,35 65x30), "OoR", text variable: rPressValue, invisible if: NOT bPressFailed
    Line (80,64) (16,35), invisible if: not bPressExcluded
    Rectangle (16,35 65x30)
        OnMouseClick:  Dialog=Dialog_DP_Field, Parameters={bSetPressExcluded: bSetPressExcluded, bSetPressIncluded: bSetPressIncluded, sHeader: sIndex}, Selected={1: , 0: }, OpenModal=True, OpenCentered=True
    Rectangle (16,35 65x30), "%2.1f Pa", text variable: rPressValue, invisible if: not bPressOffline
END_VISUALIZATION

// VISUs/Obj_Energy_Meter
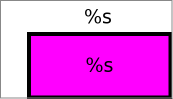
VISUALIZATION Obj_Energy_Meter  // 173x99
VAR_INPUT
	sIndex : STRING;
	bStatus : WORD;
	bOffline : BOOL;
	fOperating_Hrs : REAL;
	fEnergy : REAL;
	fVolume : REAL;
	fSupply_Temp : REAL;
	fReturn_Temp : REAL;
	fTemp_Diff :REAL;
END_VAR
    Rectangle (27,32 145x67), "%s", colour toggle: (bStatus =1) OR (bStatus = 2), text list: 'Energy_Meters_Status', text index: bStatus
        OnMouseClick:  Dialog=Dialog_EnergyMeter, Parameters={fOperHours: fOperating_Hrs, sHeader: sIndex, fTemp_Diff: fTemp_Diff, fEnergy: fEnergy, fReturn_Temp: fReturn_Temp, fSupply_Temp: fSupply_Temp, fVolume: fVolume}, OpenModal=True, OpenCentered=True
    Rectangle (23,2 150x30), "%s", text variable: sIndex
    Rectangle (27,32 145x67), "%s", invisible if: Not bOffline, text list: 'Energy_Meters_Status', text index: bStatus
END_VISUALIZATION

// VISUs/Obj_GLP_Avail
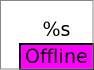
VISUALIZATION Obj_GLP_Avail  // 94x70
VAR_INPUT
	sIndex : STRING;
	bAvail : BOOL;
	bOffline : BOOL;
END_VAR
    Rectangle (19,43 75x27), "%s", text list: 'GLP_Available', text index: bAvail
    Rectangle (19,16 75x27), "%s"
    Rectangle (19,43 75x27), "Offline", invisible if: bOffline, text list: 'GLP_Status', text index: bAvail
END_VISUALIZATION

// VISUs/Obj_GLP_Status
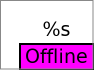
VISUALIZATION Obj_GLP_Status  // 94x70
VAR_INPUT
	sIndex : STRING;
	bAvail : BOOL;
	bOffline : BOOL;
END_VAR
    Rectangle (19,43 75x27), "%s", text list: 'GLP_Available', text index: bAvail
    Rectangle (19,16 75x27), "%s"
    Rectangle (19,43 75x27), "Offline", invisible if: bOffline, text list: 'GLP_Status', text index: bAvail
END_VISUALIZATION

// VISUs/Obj_Healthy_Failed_Field
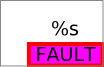
VISUALIZATION Obj_Healthy_Failed_Field  // 104x67
VAR_INPUT
	sIndex : STRING;
	bClosed : BOOL;
	bOffline : BOOL;
	bHealthy : BOOL;
END_VAR
    Rectangle (27,42 77x25), "%s", text list: 'CRAH_Isolator_Status', text index: bClosed
    Rectangle (27,16 76x26), "%s", text variable: sIndex
    Rectangle (27,42 77x25), "FAULT", invisible if: not bOffline
    Rectangle (27,42 77x25), invisible if: not bHealthy
END_VISUALIZATION

// VISUs/Obj_Leak_Detection
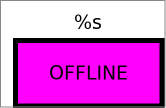
VISUALIZATION Obj_Leak_Detection  // 166x108
VAR_INPUT
	sIndex : STRING;
	bAlarm : BOOL;
	bFault : BOOL;
	bOffline : BOOL;
END_VAR
    Rectangle (13,38 151x70), "%s", colour toggle: bAlarm, text list: 'PDU_Surge_Status', text index: bAlarm
    Rectangle (13,38 151x70), "FAULT", invisible if: not bFault
    Rectangle (10,4 156x37), "%s", text variable: sIndex
    Rectangle (13,38 151x70), "OFFLINE", invisible if: not bOffline
END_VISUALIZATION

// VISUs/Obj_PDU_Breaker
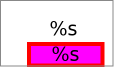
VISUALIZATION Obj_PDU_Breaker  // 114x67
VAR_INPUT
	sIndex : STRING;
	bClosed : BOOL;
	bOffline : BOOL;
	bHealthy : BOOL;
END_VAR
    Rectangle (27,42 77x25), "%s", colour toggle: bClosed, text list: 'PDU_Breaker_Status', text index: bClosed
    Rectangle (13,16 101x26), "%s", text variable: sIndex
    Rectangle (27,42 77x25), "%s", invisible if: not bOffline, text list: 'PDU_Breaker_Status', text index: bClosed
    Rectangle (27,42 77x25), invisible if: bHealthy
END_VISUALIZATION

// VISUs/Obj_PDU_Surge
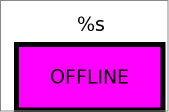
VISUALIZATION Obj_PDU_Surge  // 169x112
VAR_INPUT
	sIndex : STRING;
	bAlarm : BOOL;
	bOffline : BOOL;
END_VAR
    Rectangle (14,42 151x70), "%s", colour toggle: bAlarm, text list: 'PDU_Surge_Status', text index: bAlarm
    Rectangle (14,42 151x70), "OFFLINE", invisible if: not bOffline
    Rectangle (13,6 156x37), "%s", text variable: sIndex
END_VISUALIZATION

// VISUs/Obj_Terminal
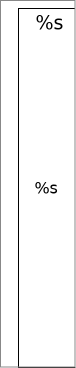
VISUALIZATION Obj_Terminal  // 76x368
VAR_INPUT
	sIndex : STRING;
	sModule : STRING;
	bOffline : BOOL;	
END_VAR
    Rectangle (18,8 57x360), "%s", text variable: sIndex, colour toggle: bOffline
    Rectangle (23,9 53x28), "%s", text variable: sModule
END_VISUALIZATION

// VISUs/Obj_THT_Field
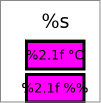
VISUALIZATION Obj_THT_Field  // 101x103
VAR_INPUT;
	rTempValue : REAL;
	rHumValue : REAL;
	bTempLimitAlarm : BOOL;
	bHumLimitAlarm : BOOL;
	bTempFailed : BOOL;
	bHumFailed : BOOL;
	bTempOffline : BOOL;
	bHumOffline : BOOL;
	bTempExcluded : BOOL;
	bHumExcluded : BOOL;
	bDeactivateDialog : BOOL;
END_VAR
    Rectangle (10,8 91x27), "%s", text variable: sIndex
    Group (25,39 60x64)
        Rectangle (0,34 60x30), "%2.1f %%", text variable: rHumValue, colour toggle: bHumLimitAlarm
        Rectangle (0,1 60x30), "%2.1f °C", text variable: rTempValue, colour toggle: bTempLimitAlarm
        Rectangle (0,0 60x30), "%2.1f °C", text variable: rTempValue, invisible if: NOT bTempExcluded
        Rectangle (0,1 60x30), "OoR", invisible if: NOT bTempFailed
        Rectangle (0,34 60x30), "%2.1f %%", text variable: rHumValue, invisible if: not bHumExcluded
        Rectangle (0,34 60x30), "OoR", invisible if: Not bHumFailed
        Line (60,30) (0,1), invisible if: not bTempExcluded
        Line (60,64) (0,35), invisible if: not bHumExcluded
        Rectangle (0,1 60x30), "%2.1f °C", text variable: rTempValue, invisible if: NOT bTempOffline
        Rectangle (0,34 60x30), "%2.1f %%", text variable: rHumValue, invisible if: NOT bHumOffline
END_VISUALIZATION

(* text list CRAH_Isolator_Status (id | default)
  0 | OFF
  1 | ON
   |  *)

(* text list CRAH_Status (id | default)
  0 | Hand
  1 | Off
  2 | Auto
   |  *)

(* text list Energy_Meters_Status (id | default)
  0 | Ok
  1 | Error
  2 | Alarm
   |  *)

(* text list Equipment_Status (id | default)
  0 | ALARM
  1 | HEALTHY
   |  *)

(* text list GLP_Available (id | default)
  0 | Not Available
  1 | Available
   |  *)

(* text list GLP_Status (id | default)
  0 | Off
  1 | On
   |  *)

(* text list Leak_Detection_Fault (id | default)
  0 | HEALTHY
  1 | FAULT
   |  *)

(* text list PDU_Breaker_Status (id | default)
  0 | Open
  1 | Closed
   |  *)

(* text list PDU_Surge_Status (id | default)
  0 | HEALTHY
  1 | ALARM
   |  *)
